// TIA Portal V15.1 export
// export: Created 2024-05-17T05:38:52.2230913Z, ExportSetting WithDefaults, DisplayName Totally Integrated Automation Portal, DisplayVersion V15.1 Update 5, DisplayName TIA Portal Openness, DisplayVersion V15.1 Update 5, DisplayName SINAMICS Startdrive Advanced, DisplayVersion V15.1, DisplayName G130, G150, S120, S150, SINAMICS MV, S210, DisplayVersion V15.1, DisplayName G110M, G120, G120C, G120D, G120P, DisplayVersion V15.1, DisplayName STEP 7 Professional, DisplayVersion V15.1 Update 5, DisplayName STEP 7 Safety, DisplayVersion V15.1, DisplayName WinCC Professional, DisplayVersion V15.1 Update 5, DisplayName SIMATIC Visualization Architect, DisplayVersion V15.1
FUNCTION_BLOCK "LGBShuttle5Pos2S-MoviFitFCPN"   // FB6696, FBD
TITLE = LGBFlinta5Pos3S-MoviFitFCPN / LGBShuttle5Pos2S-MoviFitFCPN
{ S7_Optimized_Access := 'TRUE' }
AUTHOR : VCC
VERSION : 0.0.0.0
// stored: AutoNumber false, IsIECCheckEnabled false, IsRetainMemResEnabled false, MemoryReserve 100, SetENOAutomatically False, UDAEnableTagReadback false
   VAR_INPUT
      I_Position1Begin { ExternalAccessible := 'False'; ExternalVisible := 'False'; ExternalWritable := 'False'} : Bool;   // Start Move To Position / Start Move To Position 1
      I_Position2Begin { ExternalAccessible := 'False'; ExternalVisible := 'False'; ExternalWritable := 'False'} : Bool;   // Start Move To Position / Start Move To Position 2
      I_Position3Begin { ExternalAccessible := 'False'; ExternalVisible := 'False'; ExternalWritable := 'False'} : Bool;   // Start Move To Position / Start Move To Position 3
      I_Position4Begin { ExternalAccessible := 'False'; ExternalVisible := 'False'; ExternalWritable := 'False'} : Bool;   // Start Move To Position / Start Move To Position 4
      I_Position5Begin { ExternalAccessible := 'False'; ExternalVisible := 'False'; ExternalWritable := 'False'} : Bool;   // Start Move To Position / Start Move To Position 5
      I_PositionMaintBegin { ExternalAccessible := 'False'; ExternalVisible := 'False'; ExternalWritable := 'False'} : Bool;   // Start Move To Position Maintenance
      I_SetIntlkOK { ExternalAccessible := 'False'; ExternalVisible := 'False'; ExternalWritable := 'False'} : Bool;   // Set Interlock
      I_ResIntlkOK { ExternalAccessible := 'False'; ExternalVisible := 'False'; ExternalWritable := 'False'} : Bool;   // Reset Interlock
      I_LocalPBSet { ExternalAccessible := 'False'; ExternalVisible := 'False'; ExternalWritable := 'False'} : Bool;   // Push button for manual movememt Set (on local panel)
      I_LocalPBRes { ExternalAccessible := 'False'; ExternalVisible := 'False'; ExternalWritable := 'False'} : Bool;   // Push button for manual movememt Reset (on local panel)
      I_MotorProtection { ExternalAccessible := 'False'; ExternalVisible := 'False'; ExternalWritable := 'False'} : Bool;   // Motor protection
      I_HartingPlug400V { ExternalAccessible := 'False'; ExternalVisible := 'False'; ExternalWritable := 'False'} : Bool;   // Harting plug 400V
      I_HartingPlug24V { ExternalAccessible := 'False'; ExternalVisible := 'False'; ExternalWritable := 'False'} : Bool;   // Harting plug 24V
      I_OvertravelSet { ExternalAccessible := 'False'; ExternalVisible := 'False'; ExternalWritable := 'False'} : Bool;   // Overtravel Set
      I_OvertravelRes { ExternalAccessible := 'False'; ExternalVisible := 'False'; ExternalWritable := 'False'} : Bool;   // Overtravel Reset
      I_ReferenceDet { ExternalAccessible := 'False'; ExternalVisible := 'False'; ExternalWritable := 'False'} : Bool;   // Reference detection
      I_ReleaseBrake { ExternalAccessible := 'False'; ExternalVisible := 'False'; ExternalWritable := 'False'} : Bool;   // Release brake
      I_Distance { ExternalAccessible := 'False'; ExternalVisible := 'False'; ExternalWritable := 'False'} : DInt;   // Current distance
      I_SafetyOk { ExternalAccessible := 'False'; ExternalVisible := 'False'; ExternalWritable := 'False'} : Bool;   // Safety Ok
      I_MotionStopOk { ExternalAccessible := 'False'; ExternalVisible := 'False'; ExternalWritable := 'False'} : Bool;   // The motion stop is Ok
      I_LowSpeed { ExternalAccessible := 'False'; ExternalVisible := 'False'; ExternalWritable := 'False'} : Real;   // Low speed Value (set-up %)
      I_HighSpeed { ExternalAccessible := 'False'; ExternalVisible := 'False'; ExternalWritable := 'False'} : Real;   // High speed Value (set-up %)
      I_SafetyStatusWord { ExternalAccessible := 'False'; ExternalVisible := 'False'; ExternalWritable := 'False'} : Word;   // Safety Status
      I_SafetyControlWord { ExternalAccessible := 'False'; ExternalVisible := 'False'; ExternalWritable := 'False'} : Word;   // Safety Control Word
   END_VAR
   VAR_OUTPUT
      O_ReleaseBrake { ExternalAccessible := 'False'; ExternalVisible := 'False'; ExternalWritable := 'False'} : Bool;   // Release the brake of the Motor
      O_Active { ExternalAccessible := 'False'; ExternalVisible := 'False'; ExternalWritable := 'False'} : Bool;   // Machine is active
      O_FuncRunning { ExternalAccessible := 'False'; ExternalVisible := 'False'; ExternalWritable := 'False'} : Bool;   // Signal that the function is busy
      O_InPosition1 { ExternalAccessible := 'False'; ExternalVisible := 'False'; ExternalWritable := 'False'} : Bool;   // In Position 1
      O_InPosition2 { ExternalAccessible := 'False'; ExternalVisible := 'False'; ExternalWritable := 'False'} : Bool;   // In Position 2
      O_InPosition3 { ExternalAccessible := 'False'; ExternalVisible := 'False'; ExternalWritable := 'False'} : Bool;   // In Position 3
      O_InPosition4 { ExternalAccessible := 'False'; ExternalVisible := 'False'; ExternalWritable := 'False'} : Bool;   // In Position 4
      O_InPosition5 { ExternalAccessible := 'False'; ExternalVisible := 'False'; ExternalWritable := 'False'} : Bool;   // In Position 5
      O_InPositionMaint { ExternalAccessible := 'False'; ExternalVisible := 'False'; ExternalWritable := 'False'} : Bool;   // In Position Maintenance
      O_Position1Finished { ExternalAccessible := 'False'; ExternalVisible := 'False'; ExternalWritable := 'False'} : Bool;   // Position 1 finished
      O_Position2Finished { ExternalAccessible := 'False'; ExternalVisible := 'False'; ExternalWritable := 'False'} : Bool;   // Position 2 finished
      O_Position3Finished { ExternalAccessible := 'False'; ExternalVisible := 'False'; ExternalWritable := 'False'} : Bool;   // Position 3 finished
      O_Position4Finished { ExternalAccessible := 'False'; ExternalVisible := 'False'; ExternalWritable := 'False'} : Bool;   // Position 4 finished
      O_Position5Finished { ExternalAccessible := 'False'; ExternalVisible := 'False'; ExternalWritable := 'False'} : Bool;   // Position 5 finished
      O_PositionMaintFinished { ExternalAccessible := 'False'; ExternalVisible := 'False'; ExternalWritable := 'False'} : Bool;   // Position Maintenance finished
      O_LEDPosition1 { ExternalAccessible := 'False'; ExternalVisible := 'False'; ExternalWritable := 'False'} : Bool;   // Ledindication / Led indication for Position1
      O_LEDPosition2 { ExternalAccessible := 'False'; ExternalVisible := 'False'; ExternalWritable := 'False'} : Bool;   // Ledindication / Led indication for Position2
      O_LEDPosition3 { ExternalAccessible := 'False'; ExternalVisible := 'False'; ExternalWritable := 'False'} : Bool;   // Ledindication / Led indication for Position3
      O_LEDPosition4 { ExternalAccessible := 'False'; ExternalVisible := 'False'; ExternalWritable := 'False'} : Bool;   // Ledindication / Led indication for Position4
      O_LEDPosition5 { ExternalAccessible := 'False'; ExternalVisible := 'False'; ExternalWritable := 'False'} : Bool;   // Ledindication / Led indication for Position5
      O_ReadyForOperation { ExternalAccessible := 'False'; ExternalVisible := 'False'; ExternalWritable := 'False'} : Bool;   // Ready for operation
      O_AlarmABCondition { ExternalAccessible := 'False'; ExternalVisible := 'False'; ExternalWritable := 'False'} : Bool;   // Alarm AB condition
      O_AlarmA { ExternalAccessible := 'False'; ExternalVisible := 'False'; ExternalWritable := 'False'} : Bool;   // Summation Alarm A
      O_AlarmB { ExternalAccessible := 'False'; ExternalVisible := 'False'; ExternalWritable := 'False'} : Bool;   // Summation Alarm B
      O_AlarmC { ExternalAccessible := 'False'; ExternalVisible := 'False'; ExternalWritable := 'False'} : Bool;   // Summation Alarm C
      O_AlarmD { ExternalAccessible := 'False'; ExternalVisible := 'False'; ExternalWritable := 'False'} : Bool;   // Summation Alarm D
      H_AlarmDWord { ExternalAccessible := 'False'; ExternalVisible := 'False'; ExternalWritable := 'False'} : DWord;   // HMI Animation of the alarms
      H_ActPosShuttle { ExternalAccessible := 'False'; ExternalVisible := 'False'; ExternalWritable := 'False'} : Int;   // HMI Animation Position of the Shuttle
   END_VAR
   VAR_IN_OUT
      IO_Modes : "Modes";   // Modes
      H_HMI : "H_HMI";   // Animation
      "H_GBShuttle5Pos2S-MoviFitFCPN" : "H_GBShuttle5Pos2S-MoviFitFCPN";   // Animation
      C_Config : "Shuttle5Pos2S-MoviFitFCPNConfig";   // Config
   END_VAR
   VAR
      AA_MotorProtection { ExternalAccessible := 'False'; ExternalVisible := 'False'; ExternalWritable := 'False'} : Bool;   // Motorprotection Not Ok
      AA_SafetySwitch { ExternalAccessible := 'False'; ExternalVisible := 'False'; ExternalWritable := 'False'} : Bool;   // Safety Switch Not Ok
      AB_STO { ExternalAccessible := 'False'; ExternalVisible := 'False'; ExternalWritable := 'False'} : Bool;   // Safety Switch Not Ok / Safety output to drive is active but no response from drive that the safety is ok
      AB_DriveAlarm { ExternalAccessible := 'False'; ExternalVisible := 'False'; ExternalWritable := 'False'} : Bool;   // Alarm Frequency Control
      AB_OverTravelSet { ExternalAccessible := 'False'; ExternalVisible := 'False'; ExternalWritable := 'False'} : Bool;   // Overtravel Set
      AB_OverTravelRes { ExternalAccessible := 'False'; ExternalVisible := 'False'; ExternalWritable := 'False'} : Bool;   // Overtravel Reset
      AC_KeepPos1 { ExternalAccessible := 'False'; ExternalVisible := 'False'; ExternalWritable := 'False'} : Bool;   // Lost Position 1
      AC_KeepPos2 { ExternalAccessible := 'False'; ExternalVisible := 'False'; ExternalWritable := 'False'} : Bool;   // Lost Position 2
      AC_KeepPos3 { ExternalAccessible := 'False'; ExternalVisible := 'False'; ExternalWritable := 'False'} : Bool;   // Lost Position 3
      AC_KeepPos4 { ExternalAccessible := 'False'; ExternalVisible := 'False'; ExternalWritable := 'False'} : Bool;   // Lost Position 4
      AC_KeepPos5 { ExternalAccessible := 'False'; ExternalVisible := 'False'; ExternalWritable := 'False'} : Bool;   // Lost Position 5
      AC_OvtSetAlm { ExternalAccessible := 'False'; ExternalVisible := 'False'; ExternalWritable := 'False'} : Bool;   // Timeout Set / TimeOut Set Direction
      AC_OvtResAlm { ExternalAccessible := 'False'; ExternalVisible := 'False'; ExternalWritable := 'False'} : Bool;   // Timeout Reset / TimeOut Reset Direction
      AD_IntlkSetAlm { ExternalAccessible := 'False'; ExternalVisible := 'False'; ExternalWritable := 'False'} : Bool;   // Interlock Set
      AD_IntlkResAlm { ExternalAccessible := 'False'; ExternalVisible := 'False'; ExternalWritable := 'False'} : Bool;   // Interlock Reset
      AD_OvtSetWarn { ExternalAccessible := 'False'; ExternalVisible := 'False'; ExternalWritable := 'False'} : Bool;   // TimeOut Set Direction
      AD_OvtResWarn { ExternalAccessible := 'False'; ExternalVisible := 'False'; ExternalWritable := 'False'} : Bool;   // TimeOut Reset Direction
      AD_DriveWarning { ExternalAccessible := 'False'; ExternalVisible := 'False'; ExternalWritable := 'False'} : Bool;   // Warning Frequency Control
      AA_NoBusControl { ExternalAccessible := 'False'; ExternalVisible := 'False'; ExternalWritable := 'False'} : Bool;   // Bus Control Inactive Frequency Control
      AA_HartingPlug400V { ExternalAccessible := 'False'; ExternalVisible := 'False'; ExternalWritable := 'False'} : Bool;   // Harting plug MoviFits 400VAC Not Ok
      AA_HartingPlug24V { ExternalAccessible := 'False'; ExternalVisible := 'False'; ExternalWritable := 'False'} : Bool;   // Harting plug MoviFits 24VDC Not Ok
      AB_ReferencingMode { ExternalAccessible := 'False'; ExternalVisible := 'False'; ExternalWritable := 'False'} : Bool;   // Shuttle in Referencing Mode / Flinta in Referencing Mode
      AB_NoReferencing { ExternalAccessible := 'False'; ExternalVisible := 'False'; ExternalWritable := 'False'} : Bool;   // The referencing of the Shuttle is not done. Start the Referencing procedure!
      AD_MotionStop { ExternalAccessible := 'False'; ExternalVisible := 'False'; ExternalWritable := 'False'} : Bool;   // Motion Stop
      AC_ConfigCalibrationAlm { ExternalAccessible := 'False'; ExternalVisible := 'False'; ExternalWritable := 'False'} : Bool;   // The Config values for Warming/Alarm time must be ALL zero or ALL different from zero
      AD_CalibrationWarn { ExternalAccessible := 'False'; ExternalVisible := 'False'; ExternalWritable := 'False'} : Bool;   // No High speed selected so Calibration is not possible
      AC_ConfigRampAlm { ExternalAccessible := 'False'; ExternalVisible := 'False'; ExternalWritable := 'False'} : Bool;   // The config value for the ramp is not correct, must be zero or the config values for the calculation of the ramp must be ALL zero
      AC_ConfigRampCalcAlm { ExternalAccessible := 'False'; ExternalVisible := 'False'; ExternalWritable := 'False'} : Bool;   // The config values for the calculation of the ramp must be ALL different from zero
      AD_ReferencingActive { ExternalAccessible := 'False'; ExternalVisible := 'False'; ExternalWritable := 'False'} : Bool;   // Referencing is active
      SafetyOk { ExternalAccessible := 'False'; ExternalVisible := 'False'; ExternalWritable := 'False'} : Bool;   // Safety Ok
      AlarmA { ExternalAccessible := 'False'; ExternalVisible := 'False'; ExternalWritable := 'False'} : Bool;   // Alarm A
      AlarmB { ExternalAccessible := 'False'; ExternalVisible := 'False'; ExternalWritable := 'False'} : Bool;   // Alarm B
      AlarmC { ExternalAccessible := 'False'; ExternalVisible := 'False'; ExternalWritable := 'False'} : Bool;   // Alarm C
      AlarmD { ExternalAccessible := 'False'; ExternalVisible := 'False'; ExternalWritable := 'False'} : Bool;   // Alarm D
      AlarmABCondition { ExternalAccessible := 'False'; ExternalVisible := 'False'; ExternalWritable := 'False'} : Bool;   // Alarm AB Condition
      RunTimeMaxWarn { ExternalAccessible := 'False'; ExternalVisible := 'False'; ExternalWritable := 'False'} : DInt;   // Maximum run time warning
      RunTimeMaxAlm { ExternalAccessible := 'False'; ExternalVisible := 'False'; ExternalWritable := 'False'} : DInt;   // Maximum run time alarm
      RunTimeMaxSetWarn { ExternalAccessible := 'False'; ExternalVisible := 'False'; ExternalWritable := 'False'} : DInt;   // Maximum run time warning
      RunTimeMaxSetAlm { ExternalAccessible := 'False'; ExternalVisible := 'False'; ExternalWritable := 'False'} : DInt;   // Maximum run time alarm
      RunTimeMaxResWarn { ExternalAccessible := 'False'; ExternalVisible := 'False'; ExternalWritable := 'False'} : DInt;   // Maximum run time warning
      RunTimeMaxResAlm { ExternalAccessible := 'False'; ExternalVisible := 'False'; ExternalWritable := 'False'} : DInt;   // Maximum run time alarm
      MovFuncAlmCond { ExternalAccessible := 'False'; ExternalVisible := 'False'; ExternalWritable := 'False'} : Bool;   // Move function Alarm Condition
      StopPosAlmCond { ExternalAccessible := 'False'; ExternalVisible := 'False'; ExternalWritable := 'False'} : Bool;   // Stop posistion Alarm Condition
      MotorLoopActive { ExternalAccessible := 'False'; ExternalVisible := 'False'; ExternalWritable := 'False'} : Bool;   // Motor Loop Active
      OverTravelSetAlmCond { ExternalAccessible := 'False'; ExternalVisible := 'False'; ExternalWritable := 'False'} : Bool;   // Overtravel set alarm condition
      OverTravelResAlmCond { ExternalAccessible := 'False'; ExternalVisible := 'False'; ExternalWritable := 'False'} : Bool;   // Overtravel reset alarm condition
      HartingPlug400VAlmCond { ExternalAccessible := 'False'; ExternalVisible := 'False'; ExternalWritable := 'False'} : Bool;   // Harting plug 400V alarm condition
      HartingPlug24VAlmCond { ExternalAccessible := 'False'; ExternalVisible := 'False'; ExternalWritable := 'False'} : Bool;   // Harting plug 24V alarm condition
      FuncRunning { ExternalAccessible := 'False'; ExternalVisible := 'False'; ExternalWritable := 'False'} : Bool;   // Function running
      CmdSet { ExternalAccessible := 'False'; ExternalVisible := 'False'; ExternalWritable := 'False'} : Bool;   // Command set
      CmdRes { ExternalAccessible := 'False'; ExternalVisible := 'False'; ExternalWritable := 'False'} : Bool;   // DCommand Reset
      MotorLoopAlarmCond { ExternalAccessible := 'False'; ExternalVisible := 'False'; ExternalWritable := 'False'} : Bool;   // Motor loop alarm condition
      LowerLimit { ExternalAccessible := 'False'; ExternalVisible := 'False'; ExternalWritable := 'False'} : DInt;   // Lowest position
      UpperLimit { ExternalAccessible := 'False'; ExternalVisible := 'False'; ExternalWritable := 'False'} : DInt;   // Highest position
      DiffPos { ExternalAccessible := 'False'; ExternalVisible := 'False'; ExternalWritable := 'False'} : DInt;   // Diff position
      ReferencingMode { ExternalAccessible := 'False'; ExternalVisible := 'False'; ExternalWritable := 'False'} : Bool;   // Referencing Mode
      ReferencingOvertravel { ExternalAccessible := 'False'; ExternalVisible := 'False'; ExternalWritable := 'False'} : Bool;   // During referencing mode is overtravel reached
      ReferencingFinished { ExternalAccessible := 'False'; ExternalVisible := 'False'; ExternalWritable := 'False'} : Bool;   // Referencing mode is finished
      CalculatedPos1 { ExternalAccessible := 'False'; ExternalVisible := 'False'; ExternalWritable := 'False'} : DInt;   // Calculated position 1
      CalculatedPos2 { ExternalAccessible := 'False'; ExternalVisible := 'False'; ExternalWritable := 'False'} : DInt;   // Calculated position 2
      CalculatedPos3 { ExternalAccessible := 'False'; ExternalVisible := 'False'; ExternalWritable := 'False'} : DInt;   // Calculated position 3
      CalculatedPos4 { ExternalAccessible := 'False'; ExternalVisible := 'False'; ExternalWritable := 'False'} : DInt;   // Calculated position 4
      CalculatedPos5 { ExternalAccessible := 'False'; ExternalVisible := 'False'; ExternalWritable := 'False'} : DInt;   // Calculated position 5
      CalculatedPosMaint { ExternalAccessible := 'False'; ExternalVisible := 'False'; ExternalWritable := 'False'} : DInt;   // Calculated Maintenance Position
      DirectionSetPos1 { ExternalAccessible := 'False'; ExternalVisible := 'False'; ExternalWritable := 'False'} : Bool;   // Direction SET position 1
      DirectionSetPos2 { ExternalAccessible := 'False'; ExternalVisible := 'False'; ExternalWritable := 'False'} : Bool;   // Direction SET position 2
      DirectionSetPos3 { ExternalAccessible := 'False'; ExternalVisible := 'False'; ExternalWritable := 'False'} : Bool;   // Direction SET position 3
      DirectionSetPos4 { ExternalAccessible := 'False'; ExternalVisible := 'False'; ExternalWritable := 'False'} : Bool;   // Direction SET position 4
      DirectionSetPos5 { ExternalAccessible := 'False'; ExternalVisible := 'False'; ExternalWritable := 'False'} : Bool;   // Direction SET position 5
      DirectionSetPosMaint { ExternalAccessible := 'False'; ExternalVisible := 'False'; ExternalWritable := 'False'} : Bool;   // Direction SET position Maintenance
      DirectionResPos1 { ExternalAccessible := 'False'; ExternalVisible := 'False'; ExternalWritable := 'False'} : Bool;   // Direction RESET position 1
      DirectionResPos2 { ExternalAccessible := 'False'; ExternalVisible := 'False'; ExternalWritable := 'False'} : Bool;   // Direction RESET position 2
      DirectionResPos3 { ExternalAccessible := 'False'; ExternalVisible := 'False'; ExternalWritable := 'False'} : Bool;   // Direction RESET position 3
      DirectionResPos4 { ExternalAccessible := 'False'; ExternalVisible := 'False'; ExternalWritable := 'False'} : Bool;   // Direction RESET position 4
      DirectionResPos5 { ExternalAccessible := 'False'; ExternalVisible := 'False'; ExternalWritable := 'False'} : Bool;   // Direction RESET position 5
      DirectionResPosMaint { ExternalAccessible := 'False'; ExternalVisible := 'False'; ExternalWritable := 'False'} : Bool;   // Direction RESET position Maintenance
      ManReqSetPos1 { ExternalAccessible := 'False'; ExternalVisible := 'False'; ExternalWritable := 'False'} : Bool;   // Manual request SET position 1
      ManReqSetPos2 { ExternalAccessible := 'False'; ExternalVisible := 'False'; ExternalWritable := 'False'} : Bool;   // Manual request SET position 2
      ManReqSetPos3 { ExternalAccessible := 'False'; ExternalVisible := 'False'; ExternalWritable := 'False'} : Bool;   // Manual request SET position 3
      ManReqSetPos4 { ExternalAccessible := 'False'; ExternalVisible := 'False'; ExternalWritable := 'False'} : Bool;   // Manual request SET position 4
      ManReqSetPos5 { ExternalAccessible := 'False'; ExternalVisible := 'False'; ExternalWritable := 'False'} : Bool;   // Manual request SET position 5
      ManReqSetPosMaint { ExternalAccessible := 'False'; ExternalVisible := 'False'; ExternalWritable := 'False'} : Bool;   // Manual request SET position Maintenance
      ManReqResPos1 { ExternalAccessible := 'False'; ExternalVisible := 'False'; ExternalWritable := 'False'} : Bool;   // Manual request RESET position 1
      ManReqResPos2 { ExternalAccessible := 'False'; ExternalVisible := 'False'; ExternalWritable := 'False'} : Bool;   // Manual request RESET position 2
      ManReqResPos3 { ExternalAccessible := 'False'; ExternalVisible := 'False'; ExternalWritable := 'False'} : Bool;   // Manual request RESET position 3
      ManReqResPos4 { ExternalAccessible := 'False'; ExternalVisible := 'False'; ExternalWritable := 'False'} : Bool;   // Manual request RESET position 4
      ManReqResPos5 { ExternalAccessible := 'False'; ExternalVisible := 'False'; ExternalWritable := 'False'} : Bool;   // Manual request RESET position 5
      ManReqResPosMaint { ExternalAccessible := 'False'; ExternalVisible := 'False'; ExternalWritable := 'False'} : Bool;   // Manual request RESET position Maintenance
      AutoReqSetPos1 { ExternalAccessible := 'False'; ExternalVisible := 'False'; ExternalWritable := 'False'} : Bool;   // Auto request SET position 1
      AutoReqSetPos2 { ExternalAccessible := 'False'; ExternalVisible := 'False'; ExternalWritable := 'False'} : Bool;   // Auto request SET position 2
      AutoReqSetPos3 { ExternalAccessible := 'False'; ExternalVisible := 'False'; ExternalWritable := 'False'} : Bool;   // Auto request SET position 3
      AutoReqSetPos4 { ExternalAccessible := 'False'; ExternalVisible := 'False'; ExternalWritable := 'False'} : Bool;   // Auto request SET position 4
      AutoReqSetPos5 { ExternalAccessible := 'False'; ExternalVisible := 'False'; ExternalWritable := 'False'} : Bool;   // Auto request SET position 5
      AutoReqSetPosMaint { ExternalAccessible := 'False'; ExternalVisible := 'False'; ExternalWritable := 'False'} : Bool;   // Auto request SET position Maintenance
      AutoReqResPos1 { ExternalAccessible := 'False'; ExternalVisible := 'False'; ExternalWritable := 'False'} : Bool;   // Auto request RESET position 1
      AutoReqResPos2 { ExternalAccessible := 'False'; ExternalVisible := 'False'; ExternalWritable := 'False'} : Bool;   // Auto request RESET position 2
      AutoReqResPos3 { ExternalAccessible := 'False'; ExternalVisible := 'False'; ExternalWritable := 'False'} : Bool;   // Auto request RESET position 3
      AutoReqResPos4 { ExternalAccessible := 'False'; ExternalVisible := 'False'; ExternalWritable := 'False'} : Bool;   // Auto request RESET position 4
      AutoReqResPos5 { ExternalAccessible := 'False'; ExternalVisible := 'False'; ExternalWritable := 'False'} : Bool;   // Auto request RESET position 5
      AutoReqResPosMaint { ExternalAccessible := 'False'; ExternalVisible := 'False'; ExternalWritable := 'False'} : Bool;   // Auto request RESET position Maintenance
      CmdSetPos1 { ExternalAccessible := 'False'; ExternalVisible := 'False'; ExternalWritable := 'False'} : Bool;   // Command to Position 1 in SET
      CmdSetPos2 { ExternalAccessible := 'False'; ExternalVisible := 'False'; ExternalWritable := 'False'} : Bool;   // Command to Position 2 in SET
      CmdSetPos3 { ExternalAccessible := 'False'; ExternalVisible := 'False'; ExternalWritable := 'False'} : Bool;   // Command to Position 3 in SET
      CmdSetPos4 { ExternalAccessible := 'False'; ExternalVisible := 'False'; ExternalWritable := 'False'} : Bool;   // Command to Position 4 in SET
      CmdSetPos5 { ExternalAccessible := 'False'; ExternalVisible := 'False'; ExternalWritable := 'False'} : Bool;   // Command to Position 5 in SET
      CmdSetPosMaint { ExternalAccessible := 'False'; ExternalVisible := 'False'; ExternalWritable := 'False'} : Bool;   // Command to Position Maintenance in SET
      CmdResPos1 { ExternalAccessible := 'False'; ExternalVisible := 'False'; ExternalWritable := 'False'} : Bool;   // Command to Position 1 in RESET
      CmdResPos2 { ExternalAccessible := 'False'; ExternalVisible := 'False'; ExternalWritable := 'False'} : Bool;   // Command to Position 2 in RESET
      CmdResPos3 { ExternalAccessible := 'False'; ExternalVisible := 'False'; ExternalWritable := 'False'} : Bool;   // Command to Position 3 in RESET
      CmdResPos4 { ExternalAccessible := 'False'; ExternalVisible := 'False'; ExternalWritable := 'False'} : Bool;   // Command to Position 4 in RESET
      CmdResPos5 { ExternalAccessible := 'False'; ExternalVisible := 'False'; ExternalWritable := 'False'} : Bool;   // Command to Position 5 in RESET
      CmdResPosMaint { ExternalAccessible := 'False'; ExternalVisible := 'False'; ExternalWritable := 'False'} : Bool;   // Command to Position Maintenance in RESET
      CmdPos1 { ExternalAccessible := 'False'; ExternalVisible := 'False'; ExternalWritable := 'False'} : Bool;   // Command to Position 1
      CmdPos2 { ExternalAccessible := 'False'; ExternalVisible := 'False'; ExternalWritable := 'False'} : Bool;   // Command to Position 2
      CmdPos3 { ExternalAccessible := 'False'; ExternalVisible := 'False'; ExternalWritable := 'False'} : Bool;   // Command to Position 3
      CmdPos4 { ExternalAccessible := 'False'; ExternalVisible := 'False'; ExternalWritable := 'False'} : Bool;   // Command to Position 4
      CmdPos5 { ExternalAccessible := 'False'; ExternalVisible := 'False'; ExternalWritable := 'False'} : Bool;   // Command to Position 5
      CmdPosMaint { ExternalAccessible := 'False'; ExternalVisible := 'False'; ExternalWritable := 'False'} : Bool;   // Command to Position Maintenance
      Pos1IsHomePos { ExternalAccessible := 'False'; ExternalVisible := 'False'; ExternalWritable := 'False'} : Bool;   // In position 1 / Position 1 is home position
      Pos2IsHomePos { ExternalAccessible := 'False'; ExternalVisible := 'False'; ExternalWritable := 'False'} : Bool;   // In position 2 / Position 2 is home position
      Pos3IsHomePos { ExternalAccessible := 'False'; ExternalVisible := 'False'; ExternalWritable := 'False'} : Bool;   // In position 3 / Position 3 is home position
      Pos4IsHomePos { ExternalAccessible := 'False'; ExternalVisible := 'False'; ExternalWritable := 'False'} : Bool;   // In position 4 / Position 4 is home position
      Pos5IsHomePos { ExternalAccessible := 'False'; ExternalVisible := 'False'; ExternalWritable := 'False'} : Bool;   // In position 5 / Position 5 is home position
      InPos1 { ExternalAccessible := 'False'; ExternalVisible := 'False'; ExternalWritable := 'False'} : Bool;   // In position 1
      InPos2 { ExternalAccessible := 'False'; ExternalVisible := 'False'; ExternalWritable := 'False'} : Bool;   // In position 2
      InPos3 { ExternalAccessible := 'False'; ExternalVisible := 'False'; ExternalWritable := 'False'} : Bool;   // In position 3
      InPos4 { ExternalAccessible := 'False'; ExternalVisible := 'False'; ExternalWritable := 'False'} : Bool;   // In position 4
      InPos5 { ExternalAccessible := 'False'; ExternalVisible := 'False'; ExternalWritable := 'False'} : Bool;   // In position 5
      InPosMaint { ExternalAccessible := 'False'; ExternalVisible := 'False'; ExternalWritable := 'False'} : Bool;   // In position Maintenance
      SetIntlkOK { ExternalAccessible := 'False'; ExternalVisible := 'False'; ExternalWritable := 'False'} : Bool;   // Interlock Pos1
      ResIntlkOK { ExternalAccessible := 'False'; ExternalVisible := 'False'; ExternalWritable := 'False'} : Bool;   // Interlock Pos2
      ReadyForOperation { ExternalAccessible := 'False'; ExternalVisible := 'False'; ExternalWritable := 'False'} : Bool;   // Ready for operation
      LastCmd1 { ExternalAccessible := 'False'; ExternalVisible := 'False'; ExternalWritable := 'False'} : Bool;   // Last Command to Drive Is Pos 1
      LastCmd2 { ExternalAccessible := 'False'; ExternalVisible := 'False'; ExternalWritable := 'False'} : Bool;   // Last Command to Drive Is Pos 2
      LastCmd3 { ExternalAccessible := 'False'; ExternalVisible := 'False'; ExternalWritable := 'False'} : Bool;   // Last Command to Drive Is Pos 3
      LastCmd4 { ExternalAccessible := 'False'; ExternalVisible := 'False'; ExternalWritable := 'False'} : Bool;   // Last Command to Drive Is Pos 4
      LastCmd5 { ExternalAccessible := 'False'; ExternalVisible := 'False'; ExternalWritable := 'False'} : Bool;   // Last Command to Drive Is Pos 5
      AlmCondKeepPos1 { ExternalAccessible := 'False'; ExternalVisible := 'False'; ExternalWritable := 'False'} : Bool;   // Alarm Condition Keep Position 1
      AlmCondKeepPos2 { ExternalAccessible := 'False'; ExternalVisible := 'False'; ExternalWritable := 'False'} : Bool;   // Alarm Condition Keep Position 2
      AlmCondKeepPos3 { ExternalAccessible := 'False'; ExternalVisible := 'False'; ExternalWritable := 'False'} : Bool;   // Alarm Condition Keep Position 3
      AlmCondKeepPos4 { ExternalAccessible := 'False'; ExternalVisible := 'False'; ExternalWritable := 'False'} : Bool;   // Alarm Condition Keep Position 4
      AlmCondKeepPos5 { ExternalAccessible := 'False'; ExternalVisible := 'False'; ExternalWritable := 'False'} : Bool;   // Alarm Condition Keep Position 5
      DetLowSpeedPos1 { ExternalAccessible := 'False'; ExternalVisible := 'False'; ExternalWritable := 'False'} : Bool;   // Stop high speed
      DetStopPos1 { ExternalAccessible := 'False'; ExternalVisible := 'False'; ExternalWritable := 'False'} : Bool;   // Stop on position
      DetLowSpeedPos2 { ExternalAccessible := 'False'; ExternalVisible := 'False'; ExternalWritable := 'False'} : Bool;   // Stop high speed
      DetStopPos2 { ExternalAccessible := 'False'; ExternalVisible := 'False'; ExternalWritable := 'False'} : Bool;   // Stop on position
      DetLowSpeedPos3 { ExternalAccessible := 'False'; ExternalVisible := 'False'; ExternalWritable := 'False'} : Bool;   // Stop high speed
      DetStopPos3 { ExternalAccessible := 'False'; ExternalVisible := 'False'; ExternalWritable := 'False'} : Bool;   // Stop on position
      DetLowSpeedPos4 { ExternalAccessible := 'False'; ExternalVisible := 'False'; ExternalWritable := 'False'} : Bool;   // Stop high speed
      DetStopPos4 { ExternalAccessible := 'False'; ExternalVisible := 'False'; ExternalWritable := 'False'} : Bool;   // Stop on position
      DetLowSpeedPos5 { ExternalAccessible := 'False'; ExternalVisible := 'False'; ExternalWritable := 'False'} : Bool;   // Stop high speed
      DetStopPos5 { ExternalAccessible := 'False'; ExternalVisible := 'False'; ExternalWritable := 'False'} : Bool;   // Stop on position
      DetLowSpeedPosMaint { ExternalAccessible := 'False'; ExternalVisible := 'False'; ExternalWritable := 'False'} : Bool;   // Stop high speed
      DetStopPosMaint { ExternalAccessible := 'False'; ExternalVisible := 'False'; ExternalWritable := 'False'} : Bool;   // Stop on position
      LockLocalPB { ExternalAccessible := 'False'; ExternalVisible := 'False'; ExternalWritable := 'False'} : Bool;   // Lock push button
      PODataNotEnabled { ExternalAccessible := 'False'; ExternalVisible := 'False'; ExternalWritable := 'False'} : Bool;   // Bus control inactive
      ReleaseBrake { ExternalAccessible := 'False'; ExternalVisible := 'False'; ExternalWritable := 'False'} : Bool;   // Release brake
      MotorCmdLSpdSet { ExternalAccessible := 'False'; ExternalVisible := 'False'; ExternalWritable := 'False'} : Bool;   // Command to Motorloop low Speed Set
      MotorCmdLSpdRes { ExternalAccessible := 'False'; ExternalVisible := 'False'; ExternalWritable := 'False'} : Bool;   // Command to Motorloop low speed Reset
      MotorCmdHSpdSet { ExternalAccessible := 'False'; ExternalVisible := 'False'; ExternalWritable := 'False'} : Bool;   // Command to Motorloop High Speed Set
      MotorCmdHSpdRes { ExternalAccessible := 'False'; ExternalVisible := 'False'; ExternalWritable := 'False'} : Bool;   // Command to Motorloop High Speed Reset
      PosSet { ExternalAccessible := 'False'; ExternalVisible := 'False'; ExternalWritable := 'False'} : Bool;   // Position Set detection or summary
      LowSpeedSetDet { ExternalAccessible := 'False'; ExternalVisible := 'False'; ExternalWritable := 'False'} : Bool;   // Slow Set detection or summary
      PosRes { ExternalAccessible := 'False'; ExternalVisible := 'False'; ExternalWritable := 'False'} : Bool;   // Position Reset detection or summary
      LowSpeedResDet { ExternalAccessible := 'False'; ExternalVisible := 'False'; ExternalWritable := 'False'} : Bool;   // Slow Reset detection or summary
      SetBegin { ExternalAccessible := 'False'; ExternalVisible := 'False'; ExternalWritable := 'False'} : Bool;   // Function Set begin selection
      ResBegin { ExternalAccessible := 'False'; ExternalVisible := 'False'; ExternalWritable := 'False'} : Bool;   // Function Reset begin selection
      InitDirection { ExternalAccessible := 'False'; ExternalVisible := 'False'; ExternalWritable := 'False'} : Bool;   // Initialisation of the direction
      LowSpeed { ExternalAccessible := 'False'; ExternalVisible := 'False'; ExternalWritable := 'False'} : Real;   // Low speed Value (set-up %)
      H_FncSelInHMI { ExternalAccessible := 'False'; ExternalVisible := 'False'; ExternalWritable := 'False'} : Bool;   // Function select
      H_ReferencingMode { ExternalAccessible := 'False'; ExternalVisible := 'False'; ExternalWritable := 'False'} : Bool;   // HMI Command - Activate referencing
      H_ReferencingAccept { ExternalAccessible := 'False'; ExternalVisible := 'False'; ExternalWritable := 'False'} : Bool;   // HMI Command - Reference button to accept new values
      H_CmdPos1 { ExternalAccessible := 'False'; ExternalVisible := 'False'; ExternalWritable := 'False'} : Bool;   // HMI Command - To Pos1
      H_CmdPos2 { ExternalAccessible := 'False'; ExternalVisible := 'False'; ExternalWritable := 'False'} : Bool;   // HMI Command - To Pos2
      H_CmdPos3 { ExternalAccessible := 'False'; ExternalVisible := 'False'; ExternalWritable := 'False'} : Bool;   // HMI Command - To Pos3
      H_CmdPos4 { ExternalAccessible := 'False'; ExternalVisible := 'False'; ExternalWritable := 'False'} : Bool;   // HMI Command - To Pos4
      H_CmdPos5 { ExternalAccessible := 'False'; ExternalVisible := 'False'; ExternalWritable := 'False'} : Bool;   // HMI Command - To Pos5
      H_CmdPosMaint { ExternalAccessible := 'False'; ExternalVisible := 'False'; ExternalWritable := 'False'} : Bool;   // HMI Command - To Maintenance Pos
   END_VAR
   VAR RETAIN
      H_ReferencingPos : DInt;   // Referencing position
   END_VAR
   VAR
      _SoftDetPos1 { ExternalAccessible := 'False'; ExternalVisible := 'False'; ExternalWritable := 'False'} : "LGBSoftDet";   // FB
      _SoftDetPos2 { ExternalAccessible := 'False'; ExternalVisible := 'False'; ExternalWritable := 'False'} : "LGBSoftDet";   // FB
      _SoftDetPos3 { ExternalAccessible := 'False'; ExternalVisible := 'False'; ExternalWritable := 'False'} : "LGBSoftDet";   // FB
      _SoftDetPos4 { ExternalAccessible := 'False'; ExternalVisible := 'False'; ExternalWritable := 'False'} : "LGBSoftDet";   // FB
      _SoftDetPos5 { ExternalAccessible := 'False'; ExternalVisible := 'False'; ExternalWritable := 'False'} : "LGBSoftDet";   // FB
      _SoftDetPosMaint { ExternalAccessible := 'False'; ExternalVisible := 'False'; ExternalWritable := 'False'} : "LGBSoftDet";   // FB
      _Motor { ExternalAccessible := 'False'; ExternalVisible := 'False'; ExternalWritable := 'False'} : "LGBMotor2W2S-MoviFitFCPN";   // FB
      _MovFunc2Pos2s { ExternalAccessible := 'False'; ExternalVisible := 'False'; ExternalWritable := 'False'} : "LMovFnc2Pos2S";   // FB
      _StopPos { ExternalAccessible := 'False'; ExternalVisible := 'False'; ExternalWritable := 'False'} : "L2StopPos";   // FB
      _OverTravelSet { ExternalAccessible := 'False'; ExternalVisible := 'False'; ExternalWritable := 'False'} : "L1AlarmMultiIn";   // FB
      _OverTravelRes { ExternalAccessible := 'False'; ExternalVisible := 'False'; ExternalWritable := 'False'} : "L1AlarmMultiIn";   // FB
      _HartingPlug400V { ExternalAccessible := 'False'; ExternalVisible := 'False'; ExternalWritable := 'False'} : "L1AlarmMultiIn";   // FB
      _HartingPlug24V { ExternalAccessible := 'False'; ExternalVisible := 'False'; ExternalWritable := 'False'} : "L1AlarmMultiIn";   // FB
      _KeepPositionPos1 { ExternalAccessible := 'False'; ExternalVisible := 'False'; ExternalWritable := 'False'} : "L1AlarmMultiIn";   // FB
      _KeepPositionPos2 { ExternalAccessible := 'False'; ExternalVisible := 'False'; ExternalWritable := 'False'} : "L1AlarmMultiIn";   // FB
      _KeepPositionPos3 { ExternalAccessible := 'False'; ExternalVisible := 'False'; ExternalWritable := 'False'} : "L1AlarmMultiIn";   // FB
      _KeepPositionPos4 { ExternalAccessible := 'False'; ExternalVisible := 'False'; ExternalWritable := 'False'} : "L1AlarmMultiIn";   // FB
      _KeepPositionPos5 { ExternalAccessible := 'False'; ExternalVisible := 'False'; ExternalWritable := 'False'} : "L1AlarmMultiIn";   // FB
      T_DelayPB { ExternalAccessible := 'False'; ExternalVisible := 'False'; ExternalWritable := 'False'} : TON_TIME;   // Timer
      Edge { ExternalAccessible := 'False'; ExternalVisible := 'False'; ExternalWritable := 'False'} : Array[0..20] of Bool;   // Flank
   END_VAR
   VAR_TEMP
      NotUsedH_HMI : "H_HMI";   // Animation
      H_HMIMotor : "H_HMI";   // Temp
      H_HMITemp : "H_HMI";   // Animation
      TempReal1 : Real;
      TempReal2 : Real;
      TempReal3 : Real;
   END_VAR
   VAR_TEMP   // added for the SCL form of the ladder/FBD networks
      _w1 : Bool;
      _w2 : Bool;
      _w3 : Bool;
      _w4 : Bool;
      _w5 : Bool;
   END_VAR
BEGIN

REGION Network 1: **** 1 - Inputs **** HMI Commands
   // Extract The Commands From HMI
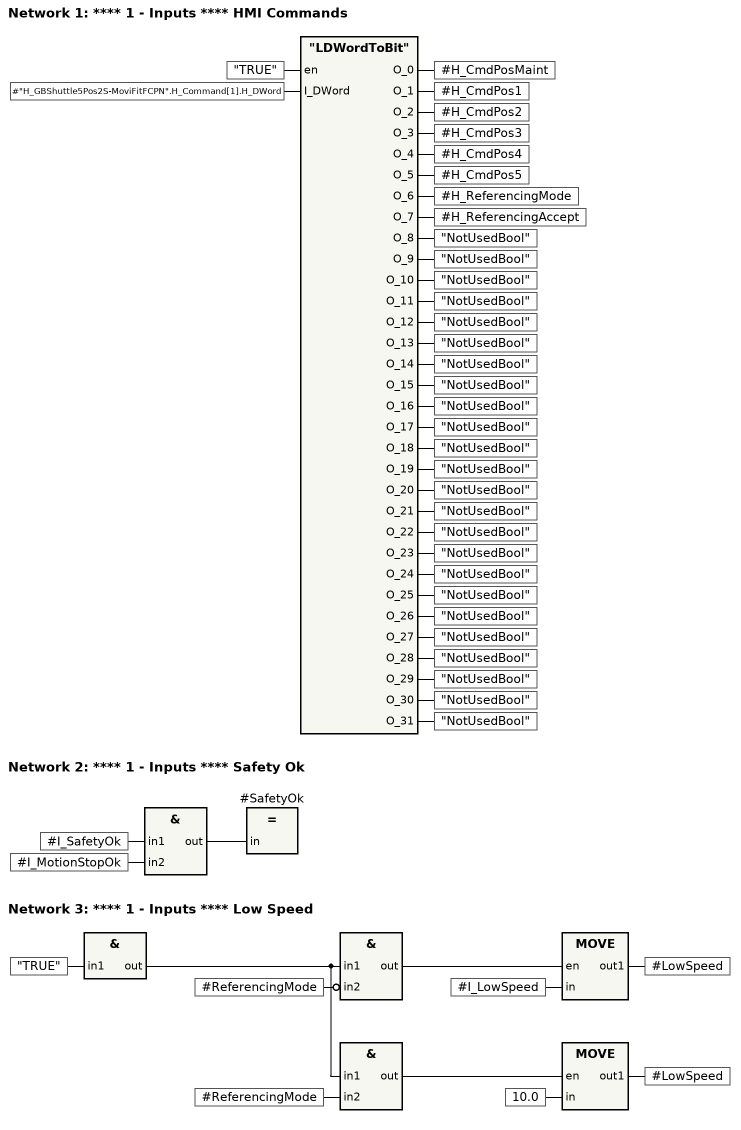
   IF "TRUE" THEN
       "LDWordToBit"(I_DWord := #"H_GBShuttle5Pos2S-MoviFitFCPN".H_Command[1].H_DWord,
                     O_0 => #H_CmdPosMaint,
                     O_1 => #H_CmdPos1,
                     O_2 => #H_CmdPos2,
                     O_3 => #H_CmdPos3,
                     O_4 => #H_CmdPos4,
                     O_5 => #H_CmdPos5,
                     O_6 => #H_ReferencingMode,
                     O_7 => #H_ReferencingAccept,
                     O_8 => "NotUsedBool",
                     O_9 => "NotUsedBool",
                     O_10 => "NotUsedBool",
                     O_11 => "NotUsedBool",
                     O_12 => "NotUsedBool",
                     O_13 => "NotUsedBool",
                     O_14 => "NotUsedBool",
                     O_15 => "NotUsedBool",
                     O_16 => "NotUsedBool",
                     O_17 => "NotUsedBool",
                     O_18 => "NotUsedBool",
                     O_19 => "NotUsedBool",
                     O_20 => "NotUsedBool",
                     O_21 => "NotUsedBool",
                     O_22 => "NotUsedBool",
                     O_23 => "NotUsedBool",
                     O_24 => "NotUsedBool",
                     O_25 => "NotUsedBool",
                     O_26 => "NotUsedBool",
                     O_27 => "NotUsedBool",
                     O_28 => "NotUsedBool",
                     O_29 => "NotUsedBool",
                     O_30 => "NotUsedBool",
                     O_31 => "NotUsedBool");
   END_IF;
END_REGION

REGION Network 2: **** 1 - Inputs **** Safety Ok
   #SafetyOk := #I_SafetyOk AND #I_MotionStopOk;
END_REGION

REGION Network 3: **** 1 - Inputs **** Low Speed
   IF "TRUE" AND NOT #ReferencingMode THEN #LowSpeed := #I_LowSpeed; END_IF;
   IF "TRUE" AND #ReferencingMode THEN #LowSpeed := 10.0; END_IF;
END_REGION

REGION Network 4: **** 1 - Inputs **** Lock local PB on position
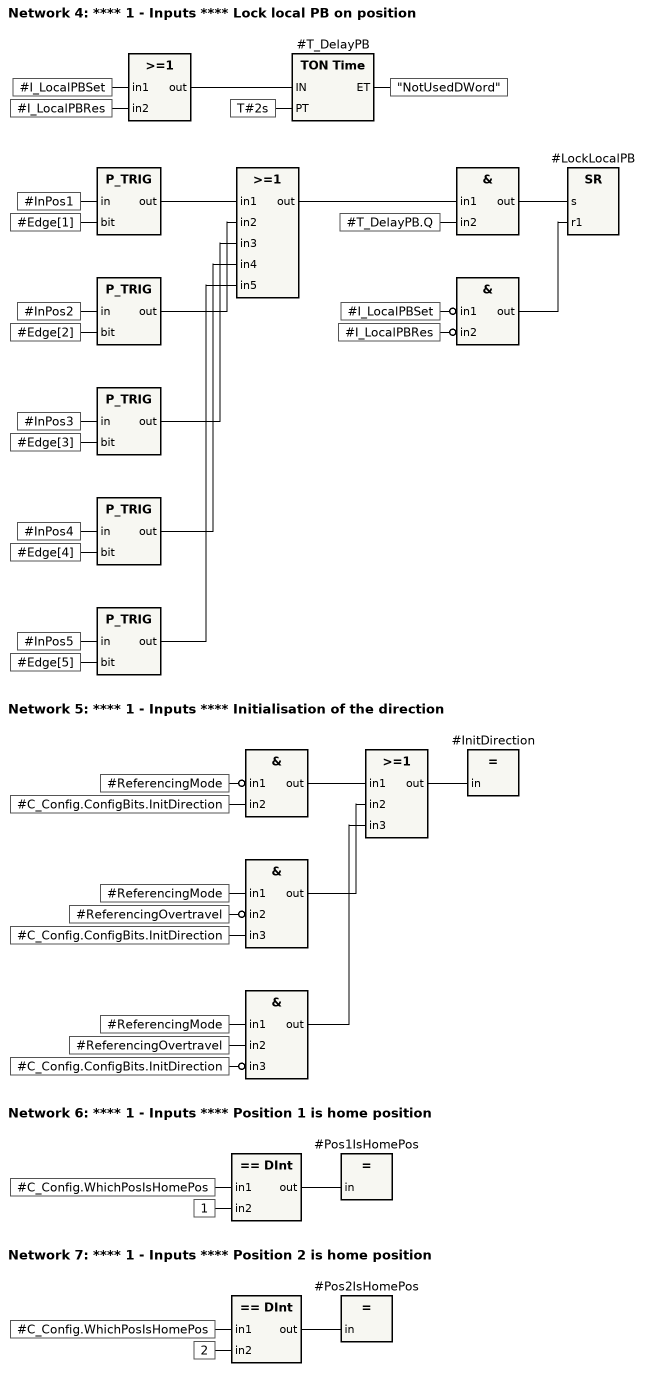
   #T_DelayPB(IN := #I_LocalPBSet OR #I_LocalPBRes, PT := T#2s, ET => "NotUsedDWord");   // TON
   #_w1 := #InPos1 AND NOT #Edge[1];   // rising edge
   #Edge[1] := #InPos1;
   #_w2 := #InPos2 AND NOT #Edge[2];   // rising edge
   #Edge[2] := #InPos2;
   #_w3 := #InPos3 AND NOT #Edge[3];   // rising edge
   #Edge[3] := #InPos3;
   #_w4 := #InPos4 AND NOT #Edge[4];   // rising edge
   #Edge[4] := #InPos4;
   #_w5 := #InPos5 AND NOT #Edge[5];   // rising edge
   #Edge[5] := #InPos5;
   IF (#_w1 OR #_w2 OR #_w3 OR #_w4 OR #_w5) AND #T_DelayPB.Q THEN
       #LockLocalPB := TRUE;   // SR flip-flop
   END_IF;
   IF NOT #I_LocalPBSet AND NOT #I_LocalPBRes THEN #LockLocalPB := FALSE; END_IF;
END_REGION

REGION Network 5: **** 1 - Inputs **** Initialisation of the direction
   #InitDirection := (NOT #ReferencingMode AND #C_Config.ConfigBits.InitDirection) OR (#ReferencingMode AND NOT #ReferencingOvertravel AND #C_Config.ConfigBits.InitDirection) OR (#ReferencingMode AND #ReferencingOvertravel AND NOT #C_Config.ConfigBits.InitDirection);
END_REGION

REGION Network 6: **** 1 - Inputs **** Position 1 is home position
   #Pos1IsHomePos := #C_Config.WhichPosIsHomePos = 1;
END_REGION

REGION Network 7: **** 1 - Inputs **** Position 2 is home position
   #Pos2IsHomePos := #C_Config.WhichPosIsHomePos = 2;
END_REGION

REGION Network 8: **** 1 - Inputs **** Position 3 is home position
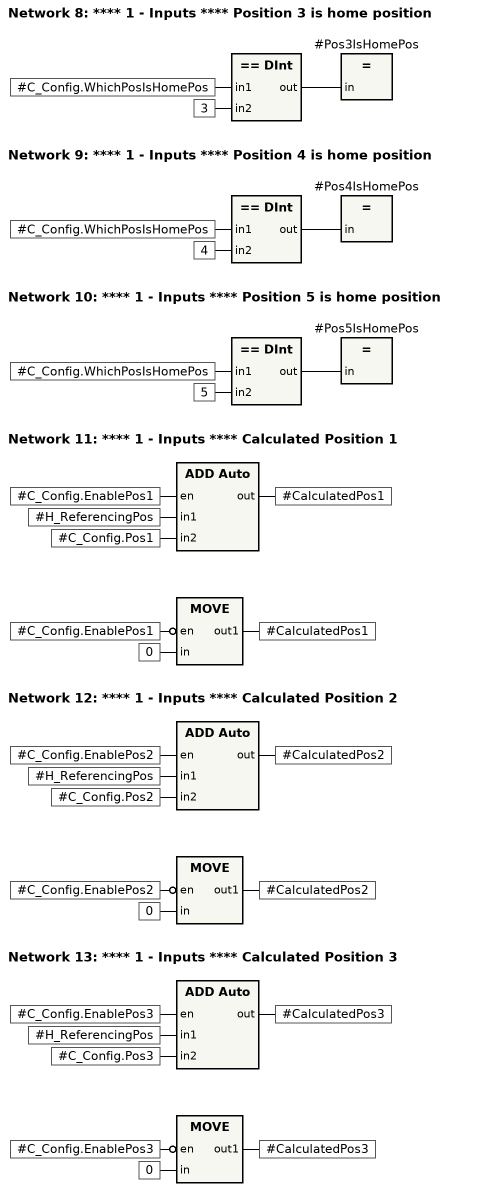
   #Pos3IsHomePos := #C_Config.WhichPosIsHomePos = 3;
END_REGION

REGION Network 9: **** 1 - Inputs **** Position 4 is home position
   #Pos4IsHomePos := #C_Config.WhichPosIsHomePos = 4;
END_REGION

REGION Network 10: **** 1 - Inputs **** Position 5 is home position
   #Pos5IsHomePos := #C_Config.WhichPosIsHomePos = 5;
END_REGION

REGION Network 11: **** 1 - Inputs **** Calculated Position 1
   IF #C_Config.EnablePos1 THEN #CalculatedPos1 := #H_ReferencingPos + #C_Config.Pos1; END_IF;
   IF NOT #C_Config.EnablePos1 THEN #CalculatedPos1 := 0; END_IF;
END_REGION

REGION Network 12: **** 1 - Inputs **** Calculated Position 2
   IF #C_Config.EnablePos2 THEN #CalculatedPos2 := #H_ReferencingPos + #C_Config.Pos2; END_IF;
   IF NOT #C_Config.EnablePos2 THEN #CalculatedPos2 := 0; END_IF;
END_REGION

REGION Network 13: **** 1 - Inputs **** Calculated Position 3
   IF #C_Config.EnablePos3 THEN #CalculatedPos3 := #H_ReferencingPos + #C_Config.Pos3; END_IF;
   IF NOT #C_Config.EnablePos3 THEN #CalculatedPos3 := 0; END_IF;
END_REGION

REGION Network 14: **** 1 - Inputs **** Calculated Position 4
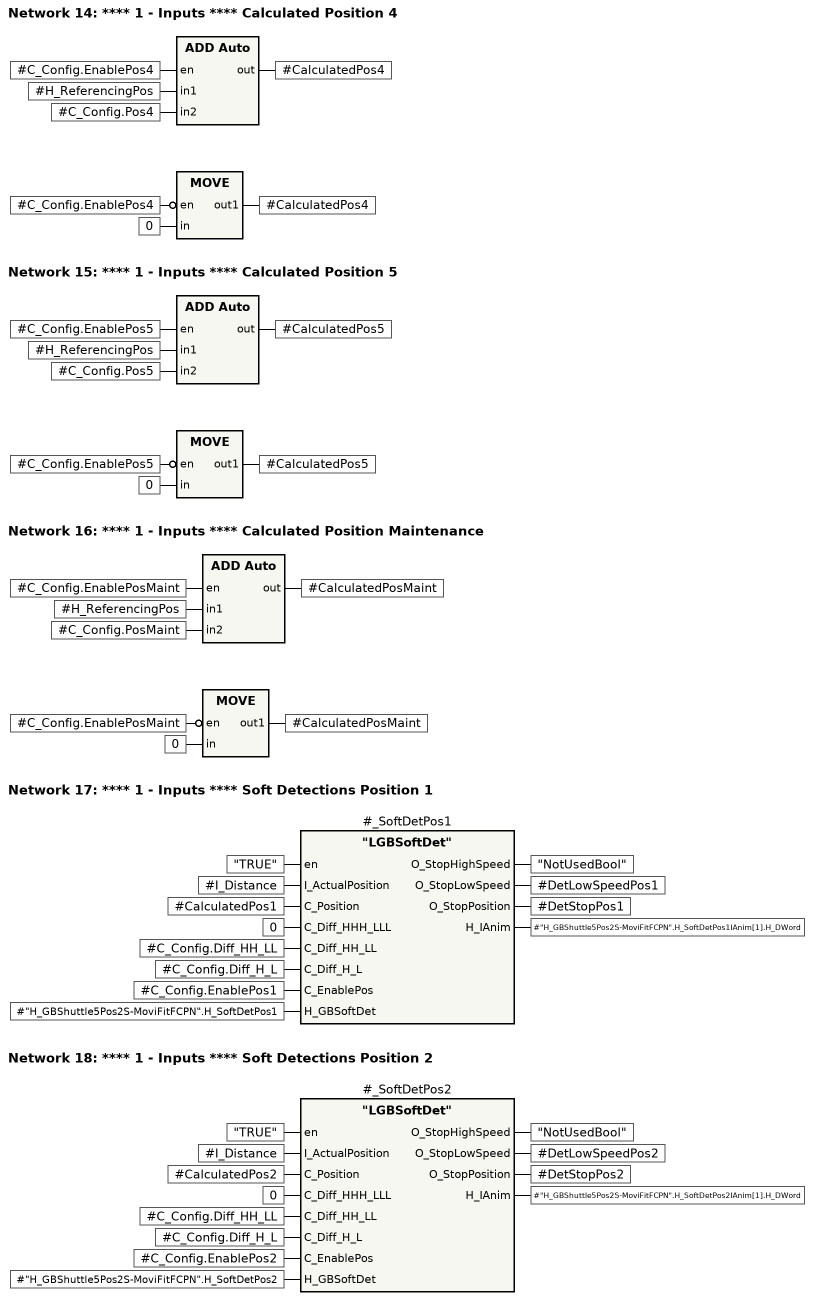
   IF #C_Config.EnablePos4 THEN #CalculatedPos4 := #H_ReferencingPos + #C_Config.Pos4; END_IF;
   IF NOT #C_Config.EnablePos4 THEN #CalculatedPos4 := 0; END_IF;
END_REGION

REGION Network 15: **** 1 - Inputs **** Calculated Position 5
   IF #C_Config.EnablePos5 THEN #CalculatedPos5 := #H_ReferencingPos + #C_Config.Pos5; END_IF;
   IF NOT #C_Config.EnablePos5 THEN #CalculatedPos5 := 0; END_IF;
END_REGION

REGION Network 16: **** 1 - Inputs **** Calculated Position Maintenance
   IF #C_Config.EnablePosMaint THEN #CalculatedPosMaint := #H_ReferencingPos + #C_Config.PosMaint; END_IF;
   IF NOT #C_Config.EnablePosMaint THEN #CalculatedPosMaint := 0; END_IF;
END_REGION

REGION Network 17: **** 1 - Inputs **** Soft Detections Position 1
   IF "TRUE" THEN
       #_SoftDetPos1(I_ActualPosition := #I_Distance,   // "LGBSoftDet"
                     C_Position := #CalculatedPos1,
                     C_Diff_HHH_LLL := 0,
                     C_Diff_HH_LL := #C_Config.Diff_HH_LL,
                     C_Diff_H_L := #C_Config.Diff_H_L,
                     C_EnablePos := #C_Config.EnablePos1,
                     H_GBSoftDet := #"H_GBShuttle5Pos2S-MoviFitFCPN".H_SoftDetPos1,
                     O_StopHighSpeed => "NotUsedBool",
                     O_StopLowSpeed => #DetLowSpeedPos1,
                     O_StopPosition => #DetStopPos1,
                     H_IAnim => #"H_GBShuttle5Pos2S-MoviFitFCPN".H_SoftDetPos1IAnim[1].H_DWord);
   END_IF;
END_REGION

REGION Network 18: **** 1 - Inputs **** Soft Detections Position 2
   IF "TRUE" THEN
       #_SoftDetPos2(I_ActualPosition := #I_Distance,   // "LGBSoftDet"
                     C_Position := #CalculatedPos2,
                     C_Diff_HHH_LLL := 0,
                     C_Diff_HH_LL := #C_Config.Diff_HH_LL,
                     C_Diff_H_L := #C_Config.Diff_H_L,
                     C_EnablePos := #C_Config.EnablePos2,
                     H_GBSoftDet := #"H_GBShuttle5Pos2S-MoviFitFCPN".H_SoftDetPos2,
                     O_StopHighSpeed => "NotUsedBool",
                     O_StopLowSpeed => #DetLowSpeedPos2,
                     O_StopPosition => #DetStopPos2,
                     H_IAnim => #"H_GBShuttle5Pos2S-MoviFitFCPN".H_SoftDetPos2IAnim[1].H_DWord);
   END_IF;
END_REGION

REGION Network 19: **** 1 - Inputs **** Soft Detections Position 3
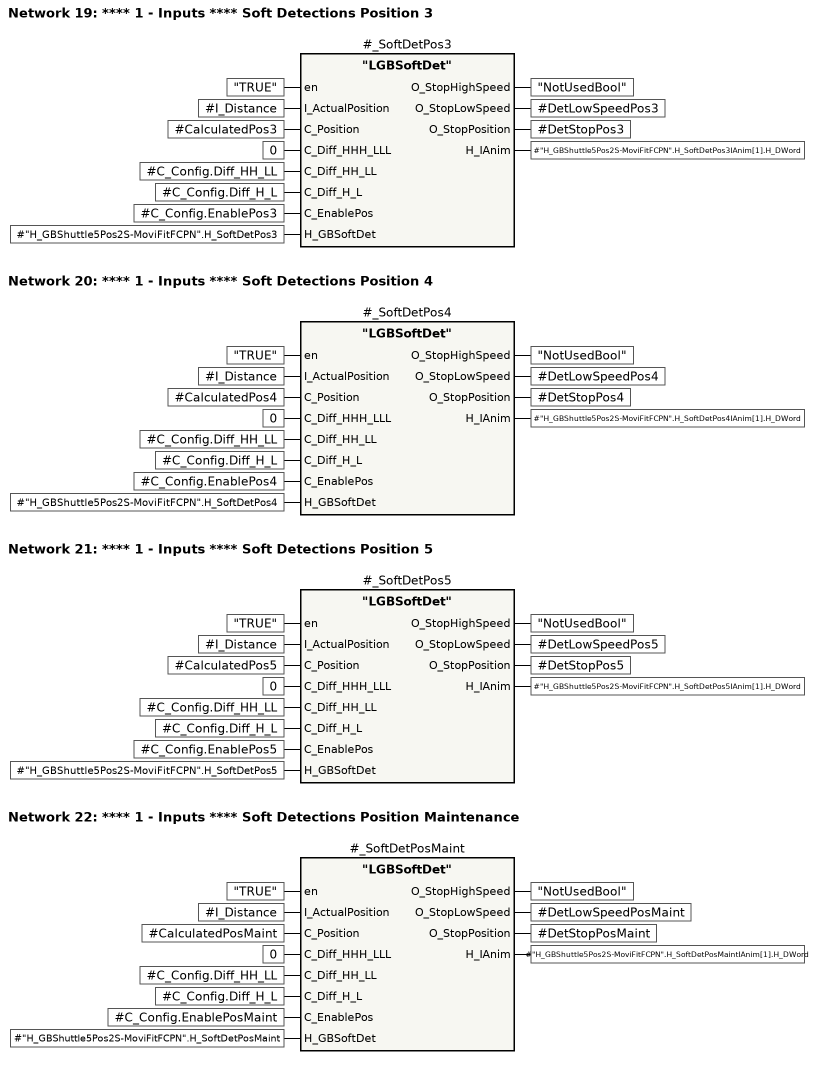
   IF "TRUE" THEN
       #_SoftDetPos3(I_ActualPosition := #I_Distance,   // "LGBSoftDet"
                     C_Position := #CalculatedPos3,
                     C_Diff_HHH_LLL := 0,
                     C_Diff_HH_LL := #C_Config.Diff_HH_LL,
                     C_Diff_H_L := #C_Config.Diff_H_L,
                     C_EnablePos := #C_Config.EnablePos3,
                     H_GBSoftDet := #"H_GBShuttle5Pos2S-MoviFitFCPN".H_SoftDetPos3,
                     O_StopHighSpeed => "NotUsedBool",
                     O_StopLowSpeed => #DetLowSpeedPos3,
                     O_StopPosition => #DetStopPos3,
                     H_IAnim => #"H_GBShuttle5Pos2S-MoviFitFCPN".H_SoftDetPos3IAnim[1].H_DWord);
   END_IF;
END_REGION

REGION Network 20: **** 1 - Inputs **** Soft Detections Position 4
   IF "TRUE" THEN
       #_SoftDetPos4(I_ActualPosition := #I_Distance,   // "LGBSoftDet"
                     C_Position := #CalculatedPos4,
                     C_Diff_HHH_LLL := 0,
                     C_Diff_HH_LL := #C_Config.Diff_HH_LL,
                     C_Diff_H_L := #C_Config.Diff_H_L,
                     C_EnablePos := #C_Config.EnablePos4,
                     H_GBSoftDet := #"H_GBShuttle5Pos2S-MoviFitFCPN".H_SoftDetPos4,
                     O_StopHighSpeed => "NotUsedBool",
                     O_StopLowSpeed => #DetLowSpeedPos4,
                     O_StopPosition => #DetStopPos4,
                     H_IAnim => #"H_GBShuttle5Pos2S-MoviFitFCPN".H_SoftDetPos4IAnim[1].H_DWord);
   END_IF;
END_REGION

REGION Network 21: **** 1 - Inputs **** Soft Detections Position 5
   IF "TRUE" THEN
       #_SoftDetPos5(I_ActualPosition := #I_Distance,   // "LGBSoftDet"
                     C_Position := #CalculatedPos5,
                     C_Diff_HHH_LLL := 0,
                     C_Diff_HH_LL := #C_Config.Diff_HH_LL,
                     C_Diff_H_L := #C_Config.Diff_H_L,
                     C_EnablePos := #C_Config.EnablePos5,
                     H_GBSoftDet := #"H_GBShuttle5Pos2S-MoviFitFCPN".H_SoftDetPos5,
                     O_StopHighSpeed => "NotUsedBool",
                     O_StopLowSpeed => #DetLowSpeedPos5,
                     O_StopPosition => #DetStopPos5,
                     H_IAnim => #"H_GBShuttle5Pos2S-MoviFitFCPN".H_SoftDetPos5IAnim[1].H_DWord);
   END_IF;
END_REGION

REGION Network 22: **** 1 - Inputs **** Soft Detections Position Maintenance
   IF "TRUE" THEN
       #_SoftDetPosMaint(I_ActualPosition := #I_Distance,   // "LGBSoftDet"
                         C_Position := #CalculatedPosMaint,
                         C_Diff_HHH_LLL := 0,
                         C_Diff_HH_LL := #C_Config.Diff_HH_LL,
                         C_Diff_H_L := #C_Config.Diff_H_L,
                         C_EnablePos := #C_Config.EnablePosMaint,
                         H_GBSoftDet := #"H_GBShuttle5Pos2S-MoviFitFCPN".H_SoftDetPosMaint,
                         O_StopHighSpeed => "NotUsedBool",
                         O_StopLowSpeed => #DetLowSpeedPosMaint,
                         O_StopPosition => #DetStopPosMaint,
                         H_IAnim => #"H_GBShuttle5Pos2S-MoviFitFCPN".H_SoftDetPosMaintIAnim[1].H_DWord);
   END_IF;
END_REGION

REGION Network 23: **** 1 - Inputs **** Direction Position 1
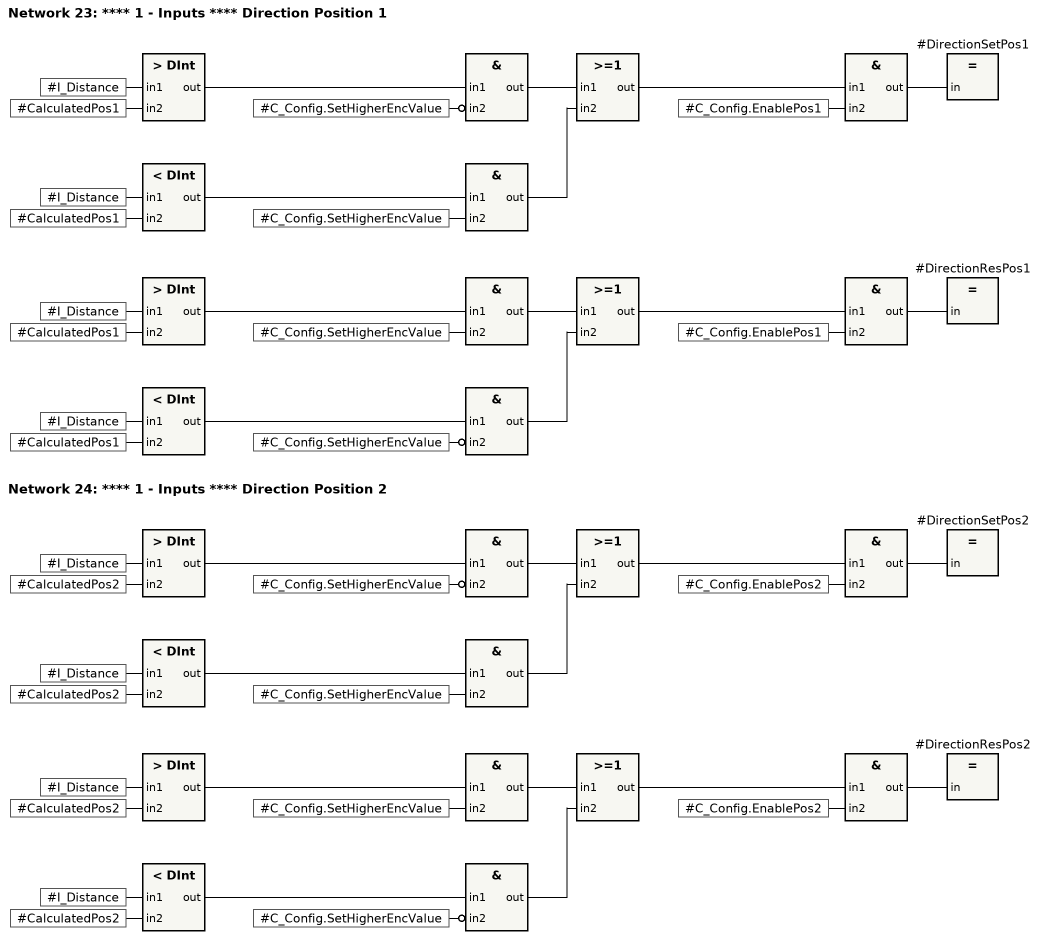
   #DirectionSetPos1 := (((#I_Distance > #CalculatedPos1) AND NOT #C_Config.SetHigherEncValue) OR ((#I_Distance < #CalculatedPos1) AND #C_Config.SetHigherEncValue)) AND #C_Config.EnablePos1;
   #DirectionResPos1 := (((#I_Distance > #CalculatedPos1) AND #C_Config.SetHigherEncValue) OR ((#I_Distance < #CalculatedPos1) AND NOT #C_Config.SetHigherEncValue)) AND #C_Config.EnablePos1;
END_REGION

REGION Network 24: **** 1 - Inputs **** Direction Position 2
   #DirectionSetPos2 := (((#I_Distance > #CalculatedPos2) AND NOT #C_Config.SetHigherEncValue) OR ((#I_Distance < #CalculatedPos2) AND #C_Config.SetHigherEncValue)) AND #C_Config.EnablePos2;
   #DirectionResPos2 := (((#I_Distance > #CalculatedPos2) AND #C_Config.SetHigherEncValue) OR ((#I_Distance < #CalculatedPos2) AND NOT #C_Config.SetHigherEncValue)) AND #C_Config.EnablePos2;
END_REGION

REGION Network 25: **** 1 - Inputs **** Direction Position 3
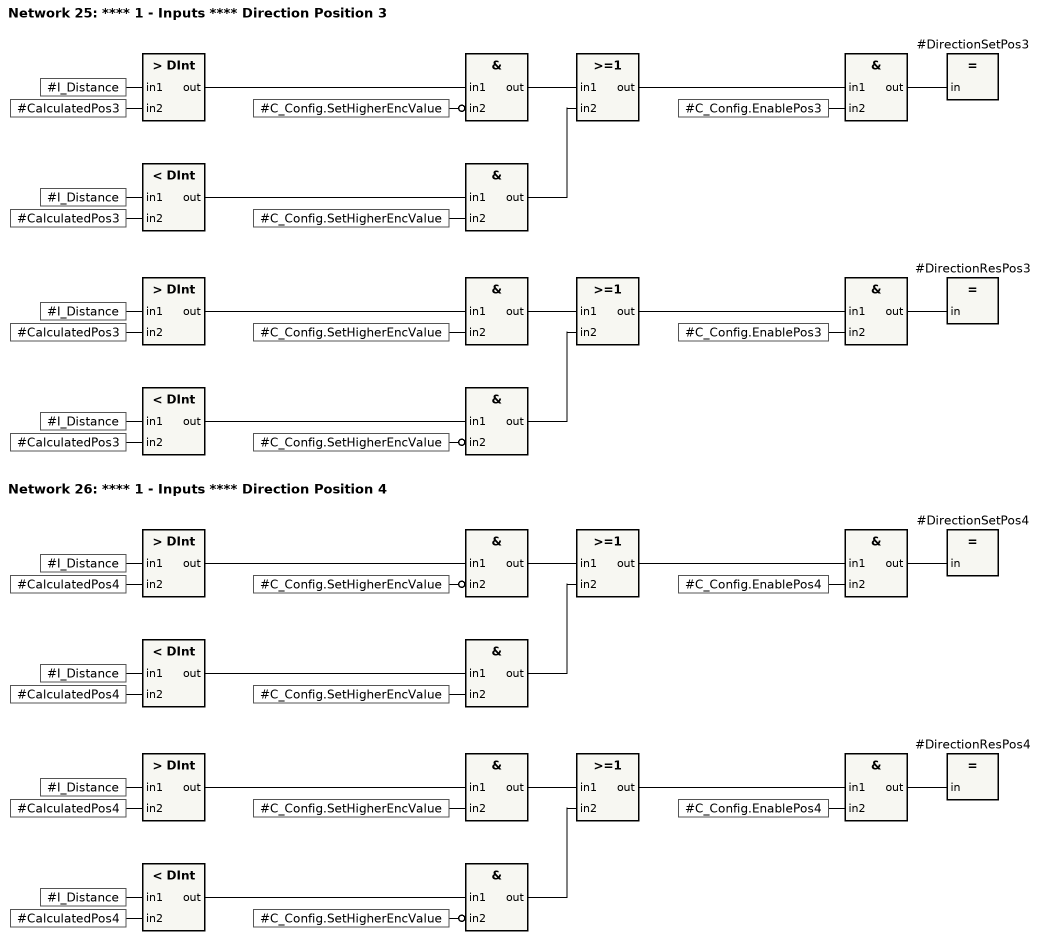
   #DirectionSetPos3 := (((#I_Distance > #CalculatedPos3) AND NOT #C_Config.SetHigherEncValue) OR ((#I_Distance < #CalculatedPos3) AND #C_Config.SetHigherEncValue)) AND #C_Config.EnablePos3;
   #DirectionResPos3 := (((#I_Distance > #CalculatedPos3) AND #C_Config.SetHigherEncValue) OR ((#I_Distance < #CalculatedPos3) AND NOT #C_Config.SetHigherEncValue)) AND #C_Config.EnablePos3;
END_REGION

REGION Network 26: **** 1 - Inputs **** Direction Position 4
   #DirectionSetPos4 := (((#I_Distance > #CalculatedPos4) AND NOT #C_Config.SetHigherEncValue) OR ((#I_Distance < #CalculatedPos4) AND #C_Config.SetHigherEncValue)) AND #C_Config.EnablePos4;
   #DirectionResPos4 := (((#I_Distance > #CalculatedPos4) AND #C_Config.SetHigherEncValue) OR ((#I_Distance < #CalculatedPos4) AND NOT #C_Config.SetHigherEncValue)) AND #C_Config.EnablePos4;
END_REGION

REGION Network 27: **** 1 - Inputs **** Direction Position 5
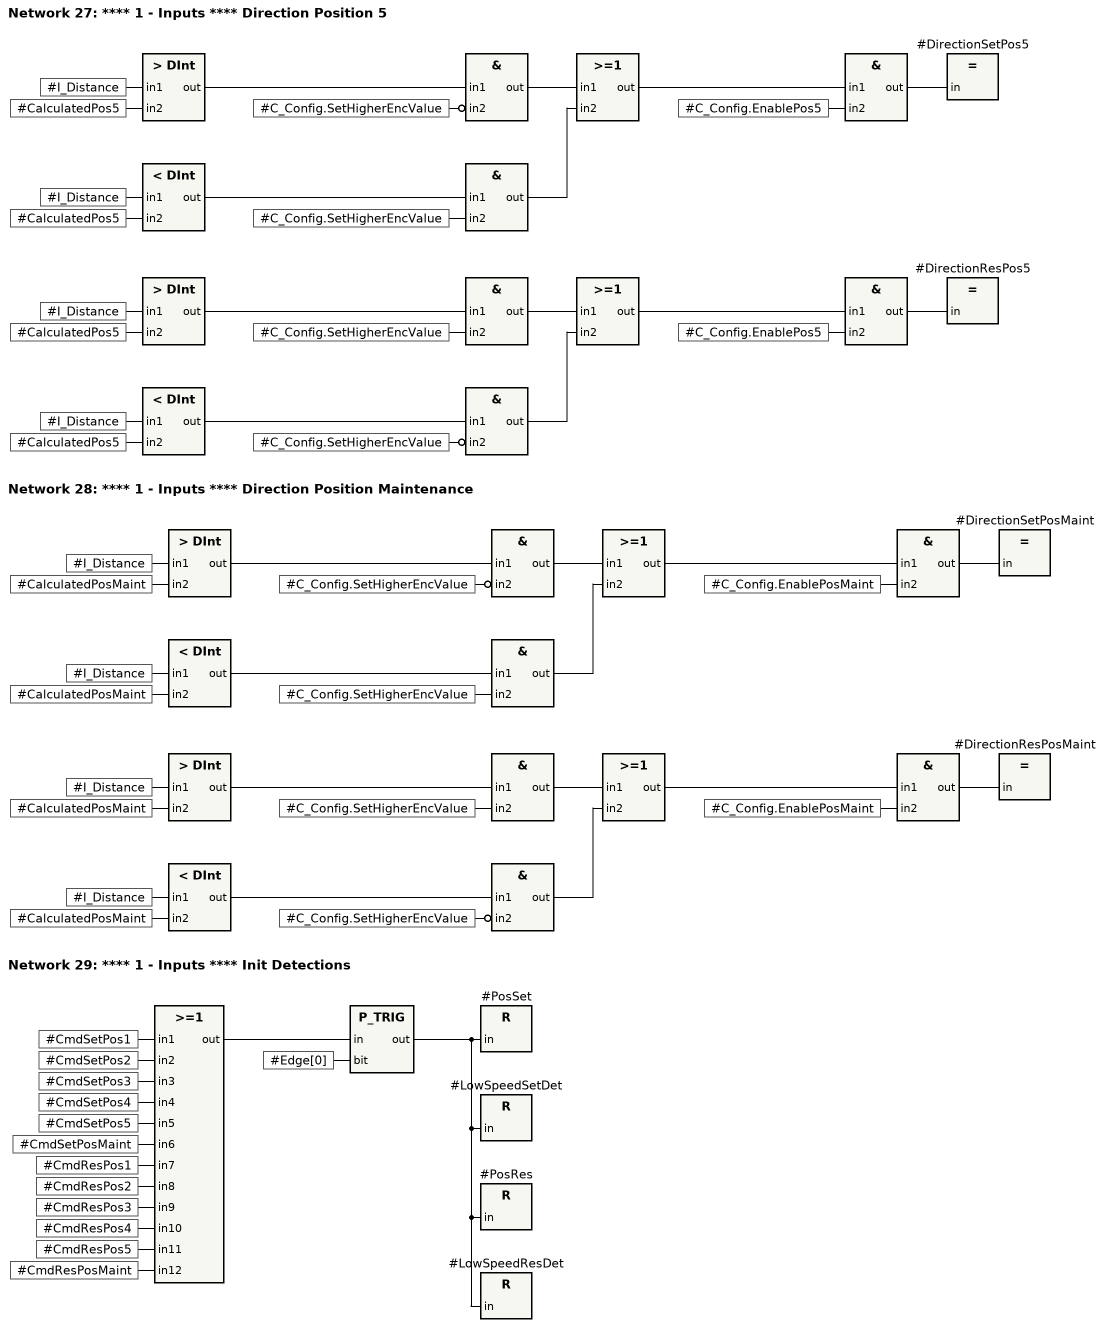
   #DirectionSetPos5 := (((#I_Distance > #CalculatedPos5) AND NOT #C_Config.SetHigherEncValue) OR ((#I_Distance < #CalculatedPos5) AND #C_Config.SetHigherEncValue)) AND #C_Config.EnablePos5;
   #DirectionResPos5 := (((#I_Distance > #CalculatedPos5) AND #C_Config.SetHigherEncValue) OR ((#I_Distance < #CalculatedPos5) AND NOT #C_Config.SetHigherEncValue)) AND #C_Config.EnablePos5;
END_REGION

REGION Network 28: **** 1 - Inputs **** Direction Position Maintenance
   #DirectionSetPosMaint := (((#I_Distance > #CalculatedPosMaint) AND NOT #C_Config.SetHigherEncValue) OR ((#I_Distance < #CalculatedPosMaint) AND #C_Config.SetHigherEncValue)) AND #C_Config.EnablePosMaint;
   #DirectionResPosMaint := (((#I_Distance > #CalculatedPosMaint) AND #C_Config.SetHigherEncValue) OR ((#I_Distance < #CalculatedPosMaint) AND NOT #C_Config.SetHigherEncValue)) AND #C_Config.EnablePosMaint;
END_REGION

REGION Network 29: **** 1 - Inputs **** Init Detections
   #_w1 := #CmdSetPos1 OR #CmdSetPos2 OR #CmdSetPos3 OR #CmdSetPos4 OR #CmdSetPos5 OR #CmdSetPosMaint OR #CmdResPos1 OR #CmdResPos2 OR #CmdResPos3 OR #CmdResPos4 OR #CmdResPos5 OR #CmdResPosMaint;
   #_w2 := #_w1 AND NOT #Edge[0];   // rising edge
   #Edge[0] := #_w1;
   IF #_w2 THEN
       #PosSet := FALSE;
       #LowSpeedSetDet := FALSE;
       #PosRes := FALSE;
       #LowSpeedResDet := FALSE;
   END_IF;
END_REGION

REGION Network 30: **** 1 - Inputs **** Detection -- Position Set
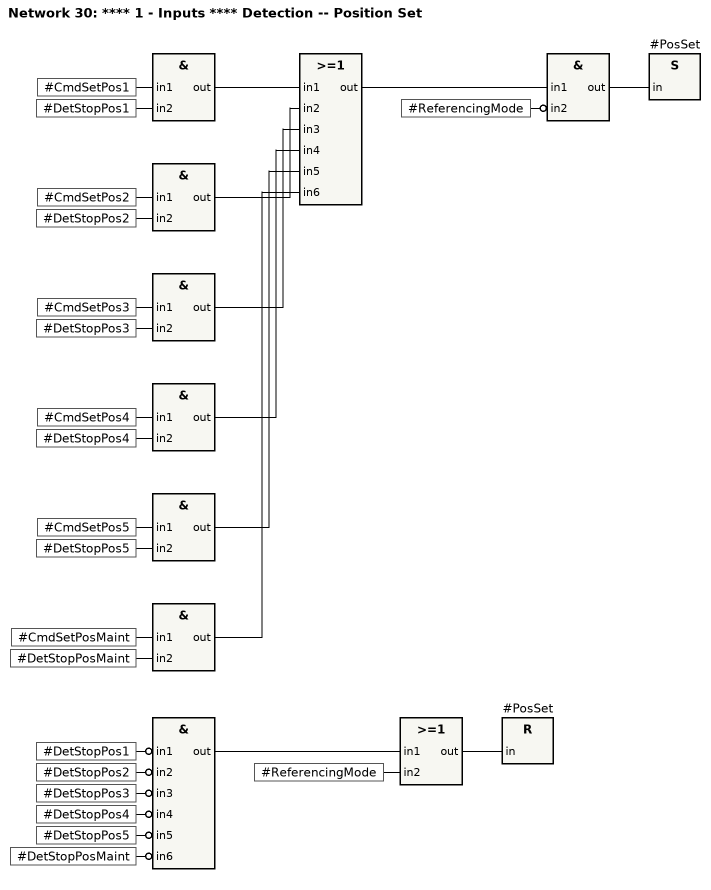
   IF ((#CmdSetPos1 AND #DetStopPos1) OR (#CmdSetPos2 AND #DetStopPos2) OR (#CmdSetPos3 AND #DetStopPos3) OR (#CmdSetPos4 AND #DetStopPos4) OR (#CmdSetPos5 AND #DetStopPos5) OR (#CmdSetPosMaint AND #DetStopPosMaint)) AND NOT #ReferencingMode THEN
       #PosSet := TRUE;
   END_IF;
   IF (NOT #DetStopPos1 AND NOT #DetStopPos2 AND NOT #DetStopPos3 AND NOT #DetStopPos4 AND NOT #DetStopPos5 AND NOT #DetStopPosMaint) OR #ReferencingMode THEN
       #PosSet := FALSE;
   END_IF;
END_REGION

REGION Network 31: **** 1 - Inputs **** Detection -- Position Set Slow
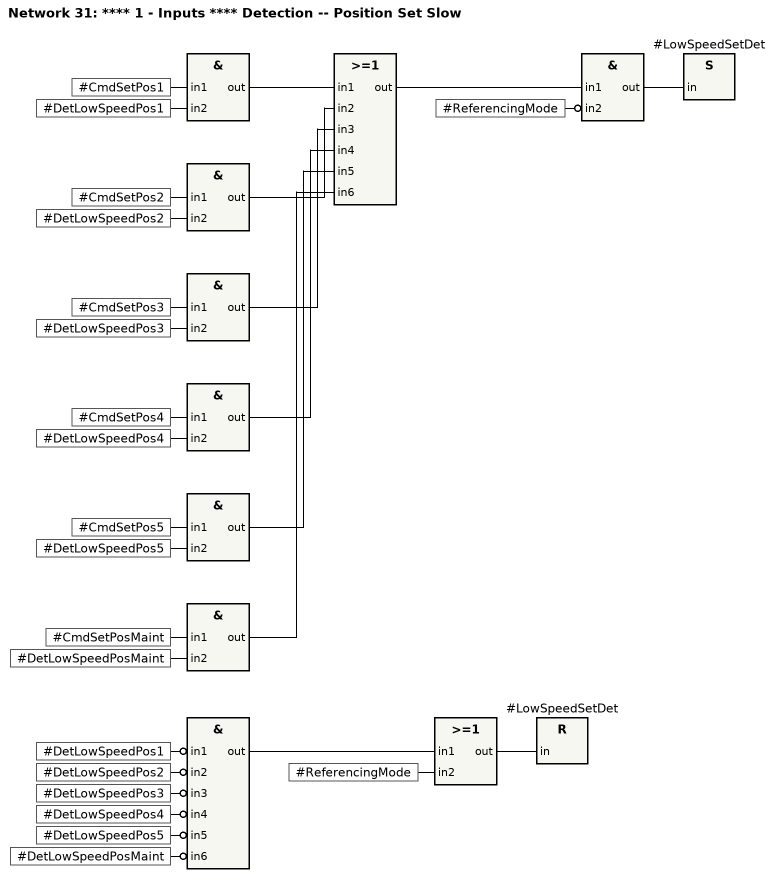
   IF ((#CmdSetPos1 AND #DetLowSpeedPos1) OR (#CmdSetPos2 AND #DetLowSpeedPos2) OR (#CmdSetPos3 AND #DetLowSpeedPos3) OR (#CmdSetPos4 AND #DetLowSpeedPos4) OR (#CmdSetPos5 AND #DetLowSpeedPos5) OR (#CmdSetPosMaint AND #DetLowSpeedPosMaint)) AND NOT #ReferencingMode THEN
       #LowSpeedSetDet := TRUE;
   END_IF;
   IF (NOT #DetLowSpeedPos1 AND NOT #DetLowSpeedPos2 AND NOT #DetLowSpeedPos3 AND NOT #DetLowSpeedPos4 AND NOT #DetLowSpeedPos5 AND NOT #DetLowSpeedPosMaint) OR #ReferencingMode THEN
       #LowSpeedSetDet := FALSE;
   END_IF;
END_REGION

REGION Network 32: **** 1 - Inputs **** Detection -- Position Reset
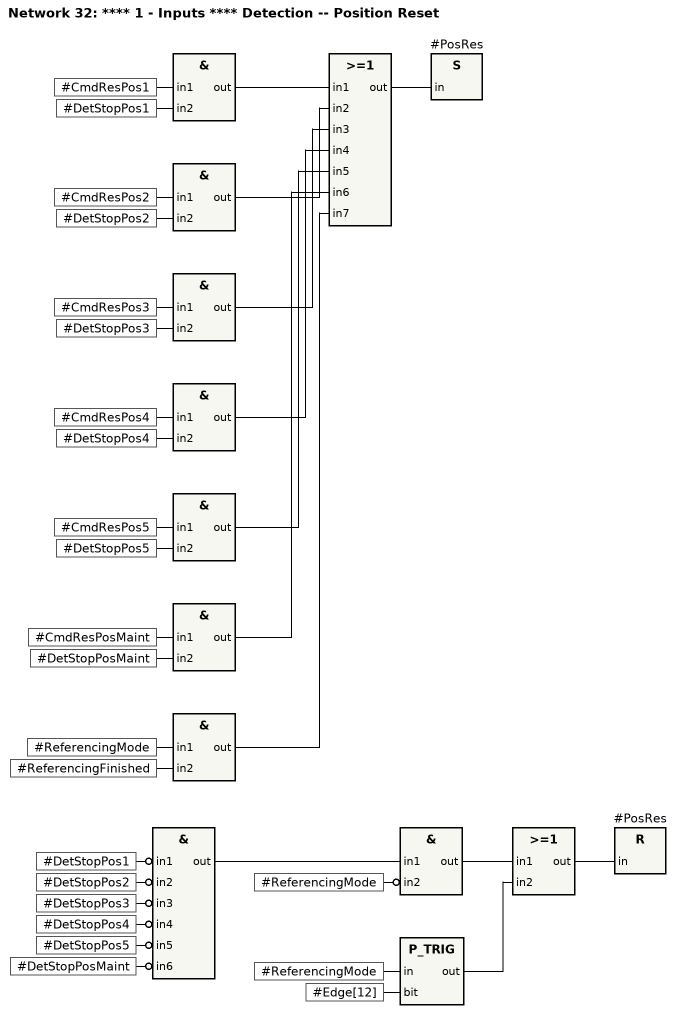
   IF (#CmdResPos1 AND #DetStopPos1) OR (#CmdResPos2 AND #DetStopPos2) OR (#CmdResPos3 AND #DetStopPos3) OR (#CmdResPos4 AND #DetStopPos4) OR (#CmdResPos5 AND #DetStopPos5) OR (#CmdResPosMaint AND #DetStopPosMaint) OR (#ReferencingMode AND #ReferencingFinished) THEN
       #PosRes := TRUE;
   END_IF;
   #_w1 := #ReferencingMode AND NOT #Edge[12];   // rising edge
   #Edge[12] := #ReferencingMode;
   IF (NOT #DetStopPos1 AND NOT #DetStopPos2 AND NOT #DetStopPos3 AND NOT #DetStopPos4 AND NOT #DetStopPos5 AND NOT #DetStopPosMaint AND NOT #ReferencingMode) OR #_w1 THEN
       #PosRes := FALSE;
   END_IF;
END_REGION

REGION Network 33: **** 1 - Inputs **** Detection -- Position Reset Slow
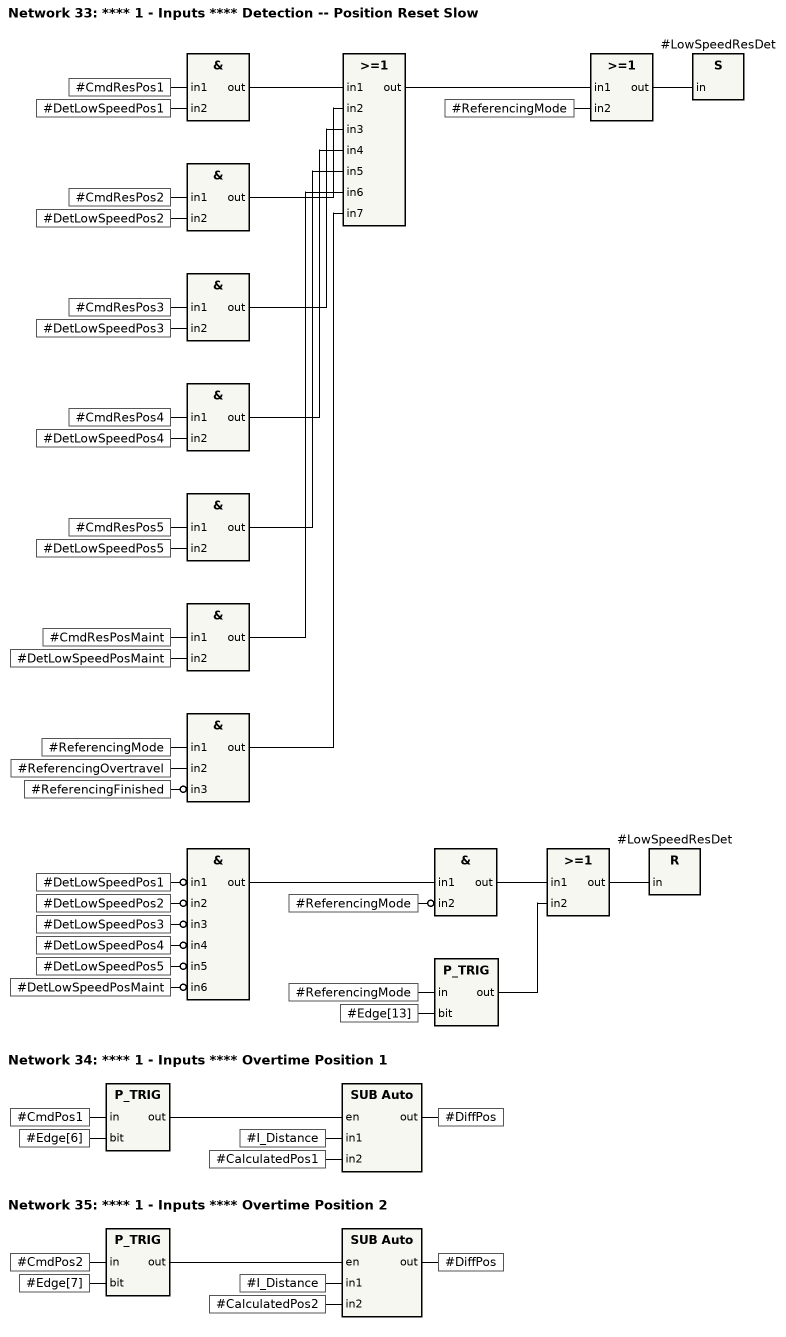
   IF (#CmdResPos1 AND #DetLowSpeedPos1) OR (#CmdResPos2 AND #DetLowSpeedPos2) OR (#CmdResPos3 AND #DetLowSpeedPos3) OR (#CmdResPos4 AND #DetLowSpeedPos4) OR (#CmdResPos5 AND #DetLowSpeedPos5) OR (#CmdResPosMaint AND #DetLowSpeedPosMaint) OR (#ReferencingMode AND #ReferencingOvertravel AND NOT #ReferencingFinished) OR #ReferencingMode THEN
       #LowSpeedResDet := TRUE;
   END_IF;
   #_w1 := #ReferencingMode AND NOT #Edge[13];   // rising edge
   #Edge[13] := #ReferencingMode;
   IF (NOT #DetLowSpeedPos1 AND NOT #DetLowSpeedPos2 AND NOT #DetLowSpeedPos3 AND NOT #DetLowSpeedPos4 AND NOT #DetLowSpeedPos5 AND NOT #DetLowSpeedPosMaint AND NOT #ReferencingMode) OR #_w1 THEN
       #LowSpeedResDet := FALSE;
   END_IF;
END_REGION

REGION Network 34: **** 1 - Inputs **** Overtime Position 1
   #_w1 := #CmdPos1 AND NOT #Edge[6];   // rising edge
   #Edge[6] := #CmdPos1;
   IF #_w1 THEN #DiffPos := #I_Distance - #CalculatedPos1; END_IF;
END_REGION

REGION Network 35: **** 1 - Inputs **** Overtime Position 2
   #_w1 := #CmdPos2 AND NOT #Edge[7];   // rising edge
   #Edge[7] := #CmdPos2;
   IF #_w1 THEN #DiffPos := #I_Distance - #CalculatedPos2; END_IF;
END_REGION

REGION Network 36: **** 1 - Inputs **** Overtime Position 3
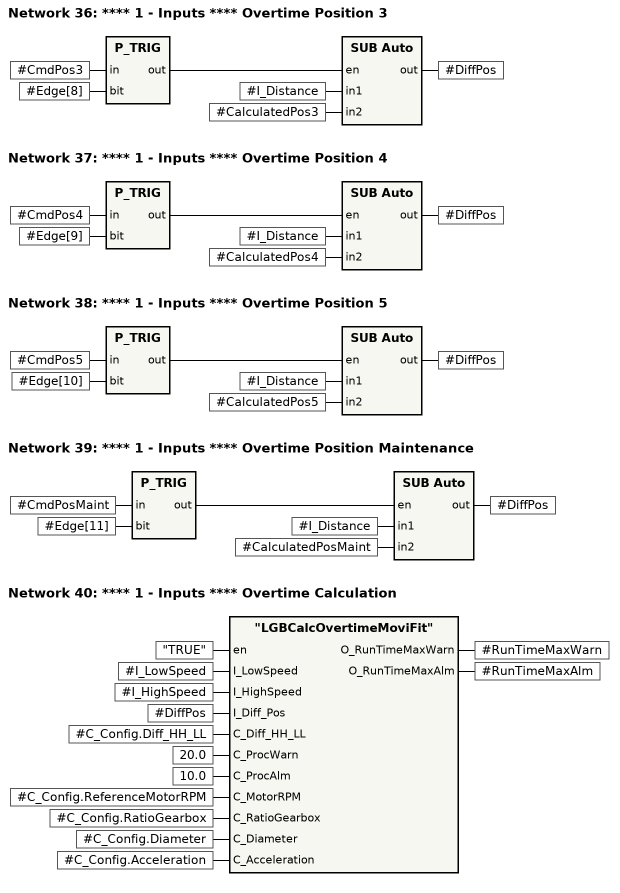
   #_w1 := #CmdPos3 AND NOT #Edge[8];   // rising edge
   #Edge[8] := #CmdPos3;
   IF #_w1 THEN #DiffPos := #I_Distance - #CalculatedPos3; END_IF;
END_REGION

REGION Network 37: **** 1 - Inputs **** Overtime Position 4
   #_w1 := #CmdPos4 AND NOT #Edge[9];   // rising edge
   #Edge[9] := #CmdPos4;
   IF #_w1 THEN #DiffPos := #I_Distance - #CalculatedPos4; END_IF;
END_REGION

REGION Network 38: **** 1 - Inputs **** Overtime Position 5
   #_w1 := #CmdPos5 AND NOT #Edge[10];   // rising edge
   #Edge[10] := #CmdPos5;
   IF #_w1 THEN #DiffPos := #I_Distance - #CalculatedPos5; END_IF;
END_REGION

REGION Network 39: **** 1 - Inputs **** Overtime Position Maintenance
   #_w1 := #CmdPosMaint AND NOT #Edge[11];   // rising edge
   #Edge[11] := #CmdPosMaint;
   IF #_w1 THEN #DiffPos := #I_Distance - #CalculatedPosMaint; END_IF;
END_REGION

REGION Network 40: **** 1 - Inputs **** Overtime Calculation
   IF "TRUE" THEN
       "LGBCalcOvertimeMoviFit"(I_LowSpeed := #I_LowSpeed,
                               I_HighSpeed := #I_HighSpeed,
                               I_Diff_Pos := #DiffPos,
                               C_Diff_HH_LL := #C_Config.Diff_HH_LL,
                               C_ProcWarn := 20.0,
                               C_ProcAlm := 10.0,
                               C_MotorRPM := #C_Config.ReferenceMotorRPM,
                               C_RatioGearbox := #C_Config.RatioGearbox,
                               C_Diameter := #C_Config.Diameter,
                               C_Acceleration := #C_Config.Acceleration,
                               O_RunTimeMaxWarn => #RunTimeMaxWarn,
                               O_RunTimeMaxAlm => #RunTimeMaxAlm);
   END_IF;
END_REGION

REGION Network 41: **** 1 - Inputs **** Overtime Result
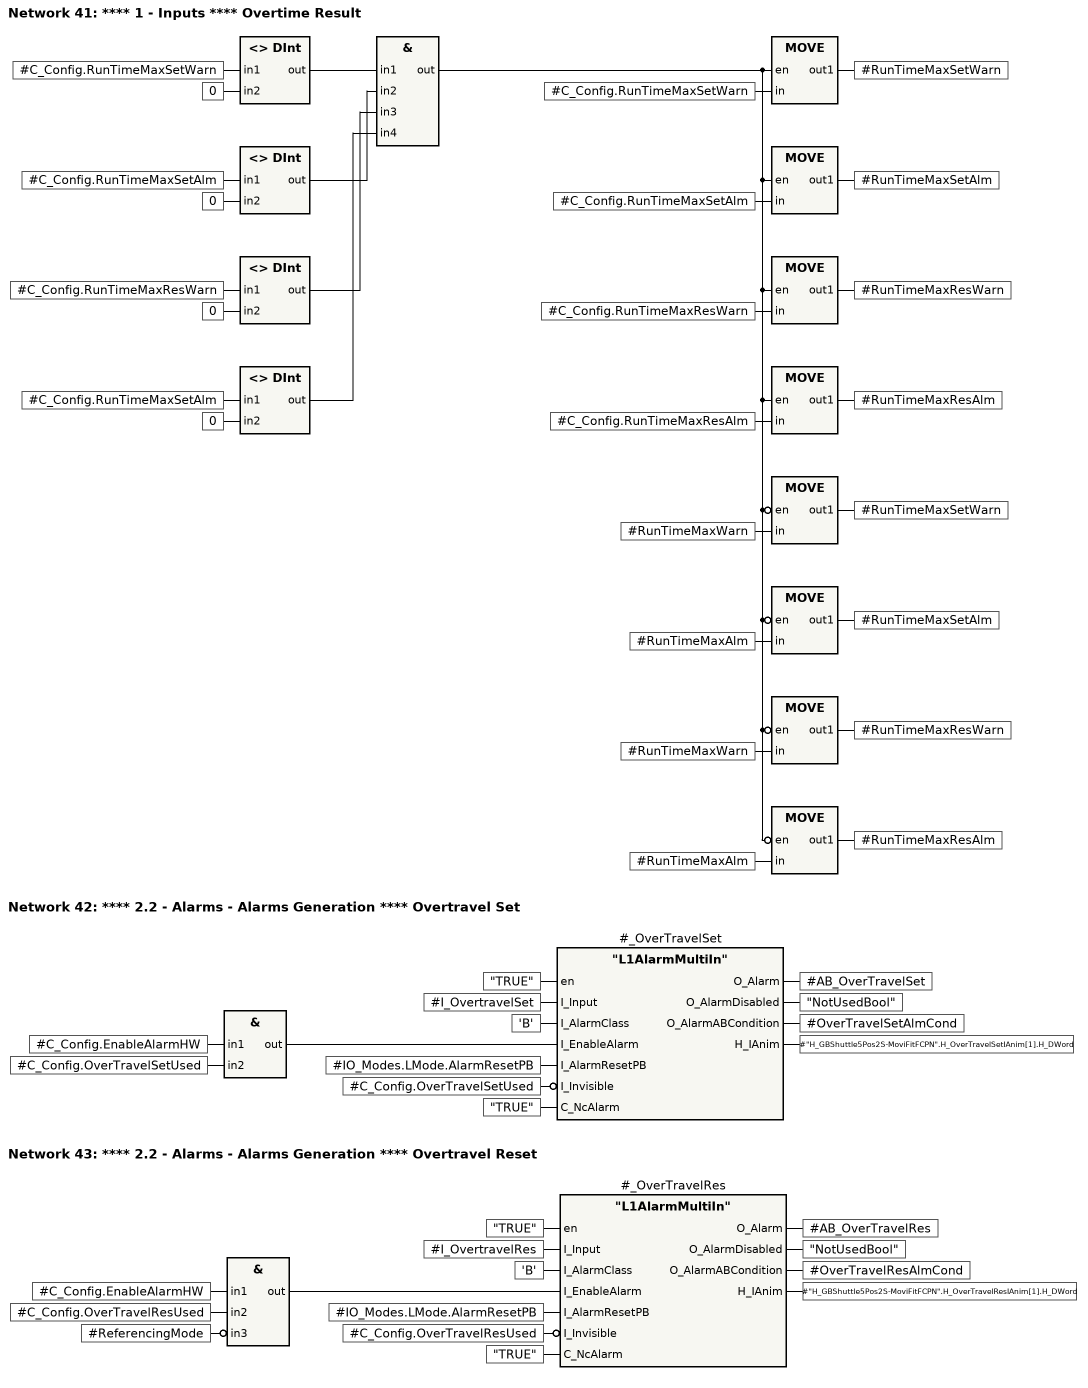
   #_w1 := (#C_Config.RunTimeMaxSetWarn <> 0) AND (#C_Config.RunTimeMaxSetAlm <> 0) AND (#C_Config.RunTimeMaxResWarn <> 0) AND (#C_Config.RunTimeMaxSetAlm <> 0);
   IF #_w1 THEN
       #RunTimeMaxSetWarn := #C_Config.RunTimeMaxSetWarn;
       #RunTimeMaxSetAlm := #C_Config.RunTimeMaxSetAlm;
       #RunTimeMaxResWarn := #C_Config.RunTimeMaxResWarn;
       #RunTimeMaxResAlm := #C_Config.RunTimeMaxResAlm;
   END_IF;
   IF NOT #_w1 THEN
       #RunTimeMaxSetWarn := #RunTimeMaxWarn;
       #RunTimeMaxSetAlm := #RunTimeMaxAlm;
       #RunTimeMaxResWarn := #RunTimeMaxWarn;
       #RunTimeMaxResAlm := #RunTimeMaxAlm;
   END_IF;
END_REGION

REGION Network 42: **** 2.2 - Alarms - Alarms Generation **** Overtravel Set
   IF "TRUE" THEN
       #_OverTravelSet(I_Input := #I_OvertravelSet,   // "L1AlarmMultiIn"
                       I_AlarmClass := 'B',
                       I_EnableAlarm := #C_Config.EnableAlarmHW AND #C_Config.OverTravelSetUsed,
                       I_AlarmResetPB := #IO_Modes.LMode.AlarmResetPB,
                       I_Invisible := NOT #C_Config.OverTravelSetUsed,
                       C_NcAlarm := "TRUE",
                       O_Alarm => #AB_OverTravelSet,
                       O_AlarmDisabled => "NotUsedBool",
                       O_AlarmABCondition => #OverTravelSetAlmCond,
                       H_IAnim => #"H_GBShuttle5Pos2S-MoviFitFCPN".H_OverTravelSetIAnim[1].H_DWord);
   END_IF;
END_REGION

REGION Network 43: **** 2.2 - Alarms - Alarms Generation **** Overtravel Reset
   IF "TRUE" THEN
       #_OverTravelRes(I_Input := #I_OvertravelRes,   // "L1AlarmMultiIn"
                       I_AlarmClass := 'B',
                       I_EnableAlarm := #C_Config.EnableAlarmHW AND #C_Config.OverTravelResUsed AND NOT #ReferencingMode,
                       I_AlarmResetPB := #IO_Modes.LMode.AlarmResetPB,
                       I_Invisible := NOT #C_Config.OverTravelResUsed,
                       C_NcAlarm := "TRUE",
                       O_Alarm => #AB_OverTravelRes,
                       O_AlarmDisabled => "NotUsedBool",
                       O_AlarmABCondition => #OverTravelResAlmCond,
                       H_IAnim => #"H_GBShuttle5Pos2S-MoviFitFCPN".H_OverTravelResIAnim[1].H_DWord);
   END_IF;
END_REGION

REGION Network 44: **** 2.2 - Alarms - Alarms Generation **** Harting plug 400VAC
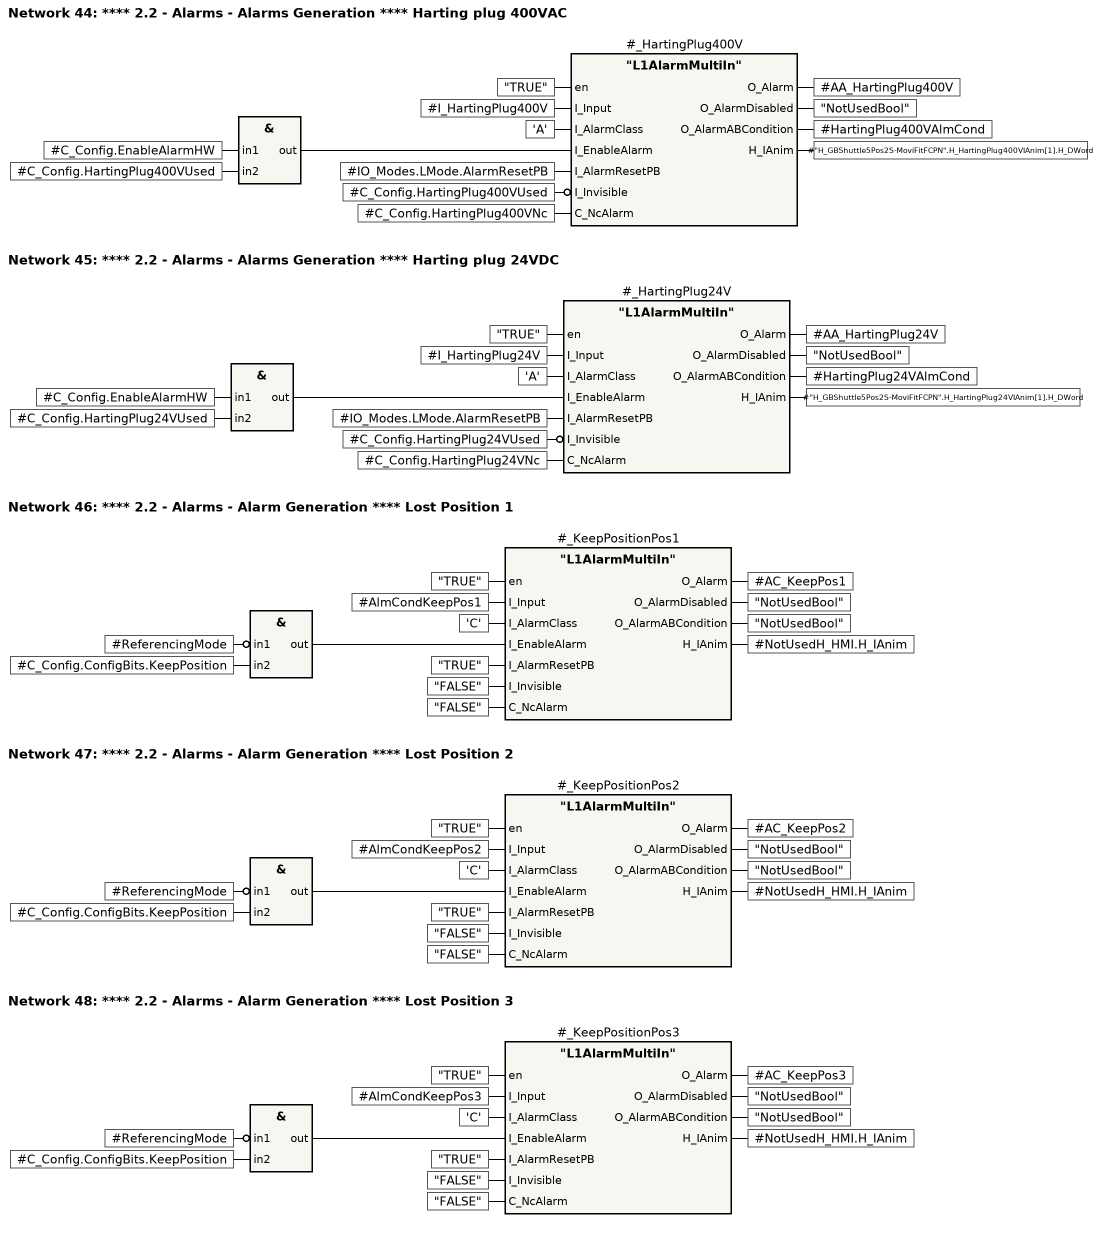
   IF "TRUE" THEN
       #_HartingPlug400V(I_Input := #I_HartingPlug400V,   // "L1AlarmMultiIn"
                         I_AlarmClass := 'A',
                         I_EnableAlarm := #C_Config.EnableAlarmHW AND #C_Config.HartingPlug400VUsed,
                         I_AlarmResetPB := #IO_Modes.LMode.AlarmResetPB,
                         I_Invisible := NOT #C_Config.HartingPlug400VUsed,
                         C_NcAlarm := #C_Config.HartingPlug400VNc,
                         O_Alarm => #AA_HartingPlug400V,
                         O_AlarmDisabled => "NotUsedBool",
                         O_AlarmABCondition => #HartingPlug400VAlmCond,
                         H_IAnim => #"H_GBShuttle5Pos2S-MoviFitFCPN".H_HartingPlug400VIAnim[1].H_DWord);
   END_IF;
END_REGION

REGION Network 45: **** 2.2 - Alarms - Alarms Generation **** Harting plug 24VDC
   IF "TRUE" THEN
       #_HartingPlug24V(I_Input := #I_HartingPlug24V,   // "L1AlarmMultiIn"
                        I_AlarmClass := 'A',
                        I_EnableAlarm := #C_Config.EnableAlarmHW AND #C_Config.HartingPlug24VUsed,
                        I_AlarmResetPB := #IO_Modes.LMode.AlarmResetPB,
                        I_Invisible := NOT #C_Config.HartingPlug24VUsed,
                        C_NcAlarm := #C_Config.HartingPlug24VNc,
                        O_Alarm => #AA_HartingPlug24V,
                        O_AlarmDisabled => "NotUsedBool",
                        O_AlarmABCondition => #HartingPlug24VAlmCond,
                        H_IAnim => #"H_GBShuttle5Pos2S-MoviFitFCPN".H_HartingPlug24VIAnim[1].H_DWord);
   END_IF;
END_REGION

REGION Network 46: **** 2.2 - Alarms - Alarm Generation **** Lost Position 1
   IF "TRUE" THEN
       #_KeepPositionPos1(I_Input := #AlmCondKeepPos1,   // "L1AlarmMultiIn"
                          I_AlarmClass := 'C',
                          I_EnableAlarm := NOT #ReferencingMode AND #C_Config.ConfigBits.KeepPosition,
                          I_AlarmResetPB := "TRUE",
                          I_Invisible := "FALSE",
                          C_NcAlarm := "FALSE",
                          O_Alarm => #AC_KeepPos1,
                          O_AlarmDisabled => "NotUsedBool",
                          O_AlarmABCondition => "NotUsedBool",
                          H_IAnim => #NotUsedH_HMI.H_IAnim);
   END_IF;
END_REGION

REGION Network 47: **** 2.2 - Alarms - Alarm Generation **** Lost Position 2
   IF "TRUE" THEN
       #_KeepPositionPos2(I_Input := #AlmCondKeepPos2,   // "L1AlarmMultiIn"
                          I_AlarmClass := 'C',
                          I_EnableAlarm := NOT #ReferencingMode AND #C_Config.ConfigBits.KeepPosition,
                          I_AlarmResetPB := "TRUE",
                          I_Invisible := "FALSE",
                          C_NcAlarm := "FALSE",
                          O_Alarm => #AC_KeepPos2,
                          O_AlarmDisabled => "NotUsedBool",
                          O_AlarmABCondition => "NotUsedBool",
                          H_IAnim => #NotUsedH_HMI.H_IAnim);
   END_IF;
END_REGION

REGION Network 48: **** 2.2 - Alarms - Alarm Generation **** Lost Position 3
   IF "TRUE" THEN
       #_KeepPositionPos3(I_Input := #AlmCondKeepPos3,   // "L1AlarmMultiIn"
                          I_AlarmClass := 'C',
                          I_EnableAlarm := NOT #ReferencingMode AND #C_Config.ConfigBits.KeepPosition,
                          I_AlarmResetPB := "TRUE",
                          I_Invisible := "FALSE",
                          C_NcAlarm := "FALSE",
                          O_Alarm => #AC_KeepPos3,
                          O_AlarmDisabled => "NotUsedBool",
                          O_AlarmABCondition => "NotUsedBool",
                          H_IAnim => #NotUsedH_HMI.H_IAnim);
   END_IF;
END_REGION

REGION Network 49: **** 2.2 - Alarms - Alarm Generation **** Lost Position 4
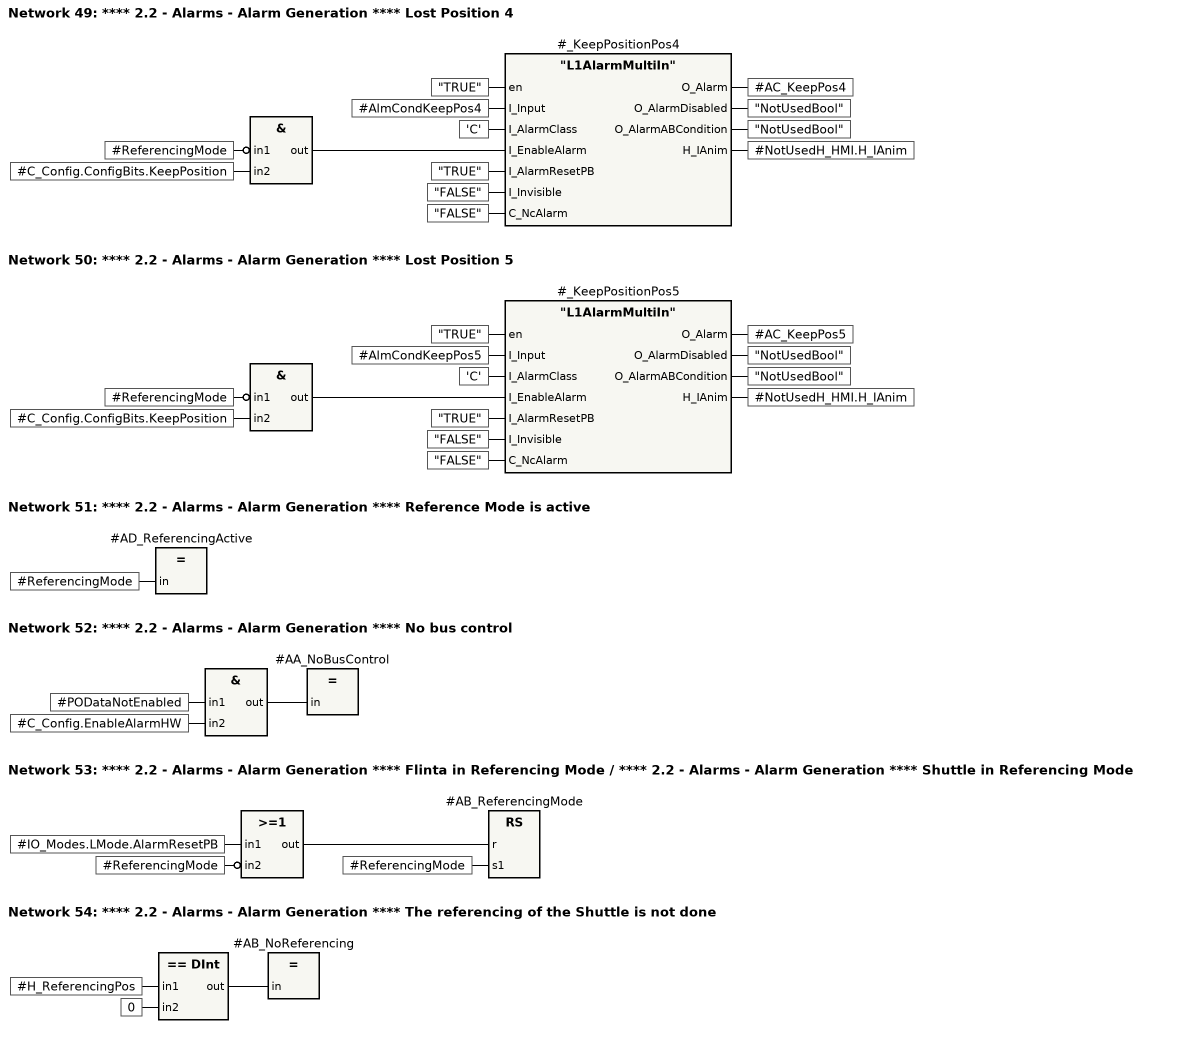
   IF "TRUE" THEN
       #_KeepPositionPos4(I_Input := #AlmCondKeepPos4,   // "L1AlarmMultiIn"
                          I_AlarmClass := 'C',
                          I_EnableAlarm := NOT #ReferencingMode AND #C_Config.ConfigBits.KeepPosition,
                          I_AlarmResetPB := "TRUE",
                          I_Invisible := "FALSE",
                          C_NcAlarm := "FALSE",
                          O_Alarm => #AC_KeepPos4,
                          O_AlarmDisabled => "NotUsedBool",
                          O_AlarmABCondition => "NotUsedBool",
                          H_IAnim => #NotUsedH_HMI.H_IAnim);
   END_IF;
END_REGION

REGION Network 50: **** 2.2 - Alarms - Alarm Generation **** Lost Position 5
   IF "TRUE" THEN
       #_KeepPositionPos5(I_Input := #AlmCondKeepPos5,   // "L1AlarmMultiIn"
                          I_AlarmClass := 'C',
                          I_EnableAlarm := NOT #ReferencingMode AND #C_Config.ConfigBits.KeepPosition,
                          I_AlarmResetPB := "TRUE",
                          I_Invisible := "FALSE",
                          C_NcAlarm := "FALSE",
                          O_Alarm => #AC_KeepPos5,
                          O_AlarmDisabled => "NotUsedBool",
                          O_AlarmABCondition => "NotUsedBool",
                          H_IAnim => #NotUsedH_HMI.H_IAnim);
   END_IF;
END_REGION

REGION Network 51: **** 2.2 - Alarms - Alarm Generation **** Reference Mode is active
   #AD_ReferencingActive := #ReferencingMode;
END_REGION

REGION Network 52: **** 2.2 - Alarms - Alarm Generation **** No bus control
   #AA_NoBusControl := #PODataNotEnabled AND #C_Config.EnableAlarmHW;
END_REGION

REGION Network 53: **** 2.2 - Alarms - Alarm Generation **** Flinta in Referencing Mode / **** 2.2 - Alarms - Alarm Generation **** Shuttle in Referencing Mode
   IF #IO_Modes.LMode.AlarmResetPB OR NOT #ReferencingMode THEN
       #AB_ReferencingMode := FALSE;   // RS flip-flop
   END_IF;
   IF #ReferencingMode THEN #AB_ReferencingMode := TRUE; END_IF;
END_REGION

REGION Network 54: **** 2.2 - Alarms - Alarm Generation **** The referencing of the Shuttle is not done
   #AB_NoReferencing := #H_ReferencingPos = 0;
END_REGION

REGION Network 55: **** 4.3 - Machine status - Operator Selection **** Manual request position 1
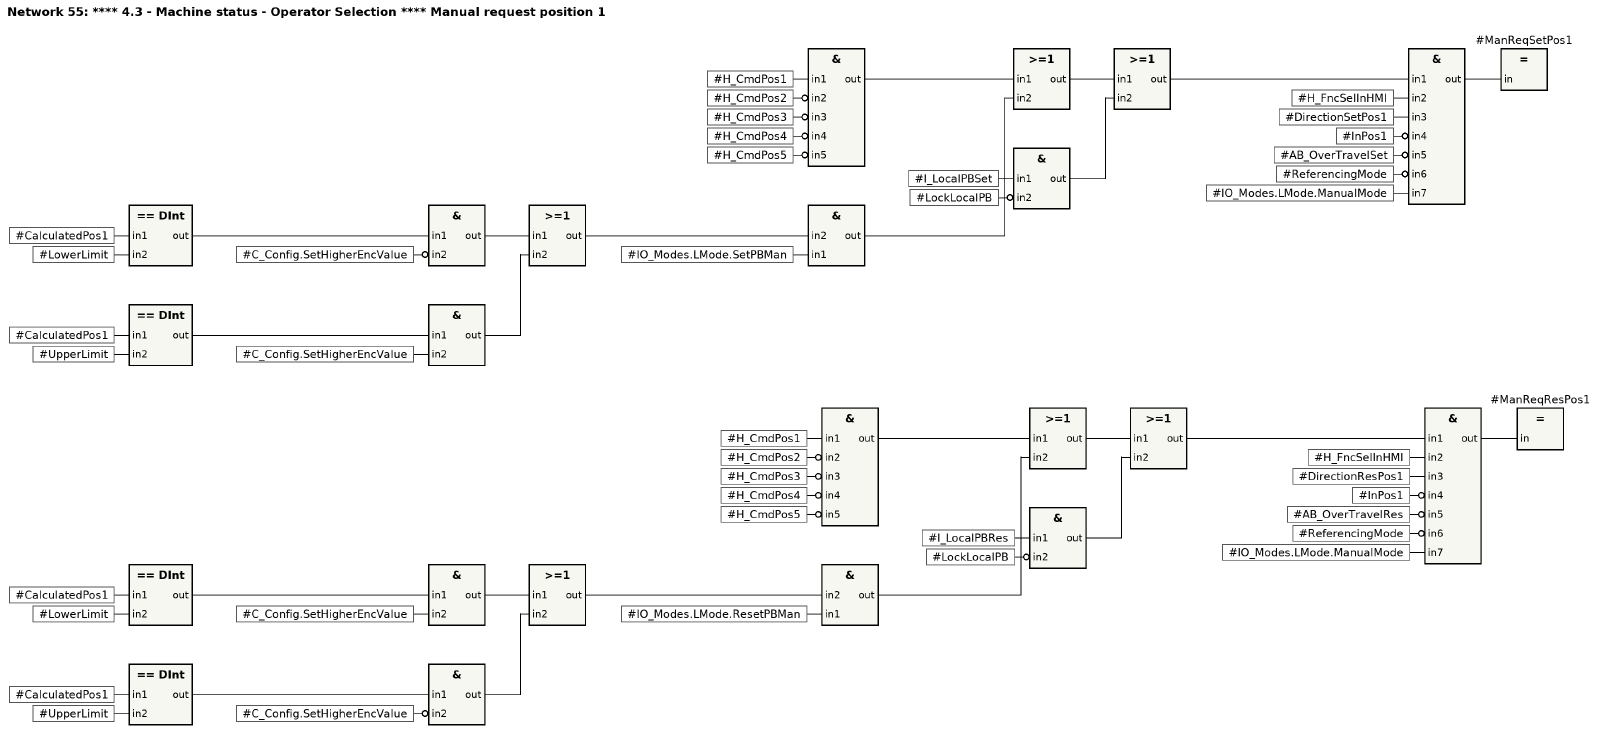
   #ManReqSetPos1 := ((#H_CmdPos1 AND NOT #H_CmdPos2 AND NOT #H_CmdPos3 AND NOT #H_CmdPos4 AND NOT #H_CmdPos5) OR ((((#CalculatedPos1 = #LowerLimit) AND NOT #C_Config.SetHigherEncValue) OR ((#CalculatedPos1 = #UpperLimit) AND #C_Config.SetHigherEncValue)) AND #IO_Modes.LMode.SetPBMan) OR (#I_LocalPBSet AND NOT #LockLocalPB)) AND #H_FncSelInHMI AND #DirectionSetPos1 AND NOT #InPos1 AND NOT #AB_OverTravelSet AND NOT #ReferencingMode AND #IO_Modes.LMode.ManualMode;
   #ManReqResPos1 := ((#H_CmdPos1 AND NOT #H_CmdPos2 AND NOT #H_CmdPos3 AND NOT #H_CmdPos4 AND NOT #H_CmdPos5) OR ((((#CalculatedPos1 = #LowerLimit) AND #C_Config.SetHigherEncValue) OR ((#CalculatedPos1 = #UpperLimit) AND NOT #C_Config.SetHigherEncValue)) AND #IO_Modes.LMode.ResetPBMan) OR (#I_LocalPBRes AND NOT #LockLocalPB)) AND #H_FncSelInHMI AND #DirectionResPos1 AND NOT #InPos1 AND NOT #AB_OverTravelRes AND NOT #ReferencingMode AND #IO_Modes.LMode.ManualMode;
END_REGION

REGION Network 56: **** 4.3 - Machine status - Operator Selection **** Manual request position 2
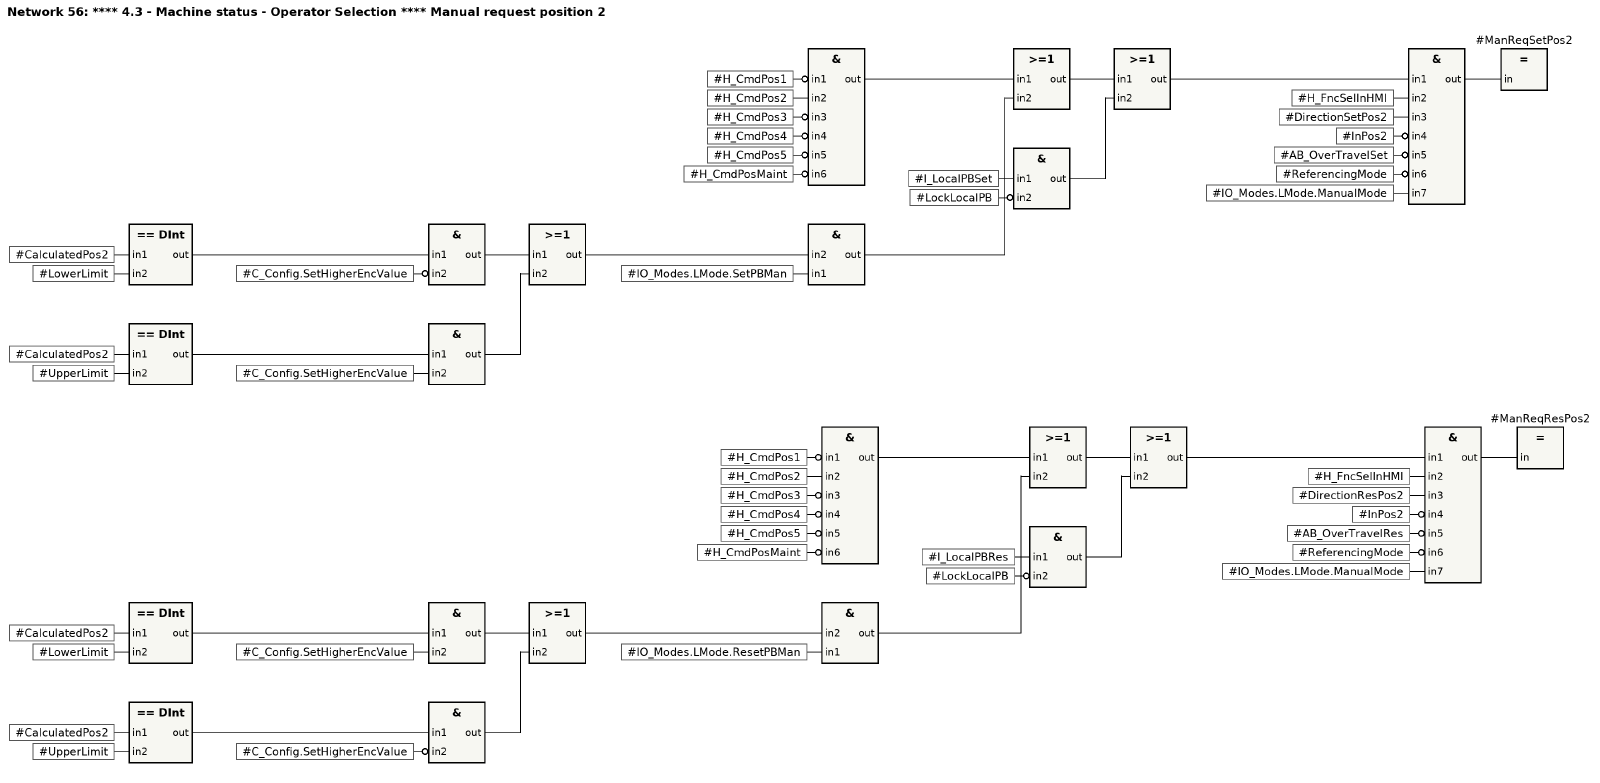
   #ManReqSetPos2 := ((NOT #H_CmdPos1 AND #H_CmdPos2 AND NOT #H_CmdPos3 AND NOT #H_CmdPos4 AND NOT #H_CmdPos5 AND NOT #H_CmdPosMaint) OR ((((#CalculatedPos2 = #LowerLimit) AND NOT #C_Config.SetHigherEncValue) OR ((#CalculatedPos2 = #UpperLimit) AND #C_Config.SetHigherEncValue)) AND #IO_Modes.LMode.SetPBMan) OR (#I_LocalPBSet AND NOT #LockLocalPB)) AND #H_FncSelInHMI AND #DirectionSetPos2 AND NOT #InPos2 AND NOT #AB_OverTravelSet AND NOT #ReferencingMode AND #IO_Modes.LMode.ManualMode;
   #ManReqResPos2 := ((NOT #H_CmdPos1 AND #H_CmdPos2 AND NOT #H_CmdPos3 AND NOT #H_CmdPos4 AND NOT #H_CmdPos5 AND NOT #H_CmdPosMaint) OR ((((#CalculatedPos2 = #LowerLimit) AND #C_Config.SetHigherEncValue) OR ((#CalculatedPos2 = #UpperLimit) AND NOT #C_Config.SetHigherEncValue)) AND #IO_Modes.LMode.ResetPBMan) OR (#I_LocalPBRes AND NOT #LockLocalPB)) AND #H_FncSelInHMI AND #DirectionResPos2 AND NOT #InPos2 AND NOT #AB_OverTravelRes AND NOT #ReferencingMode AND #IO_Modes.LMode.ManualMode;
END_REGION

REGION Network 57: **** 4.3 - Machine status - Operator Selection **** Manual request position 3
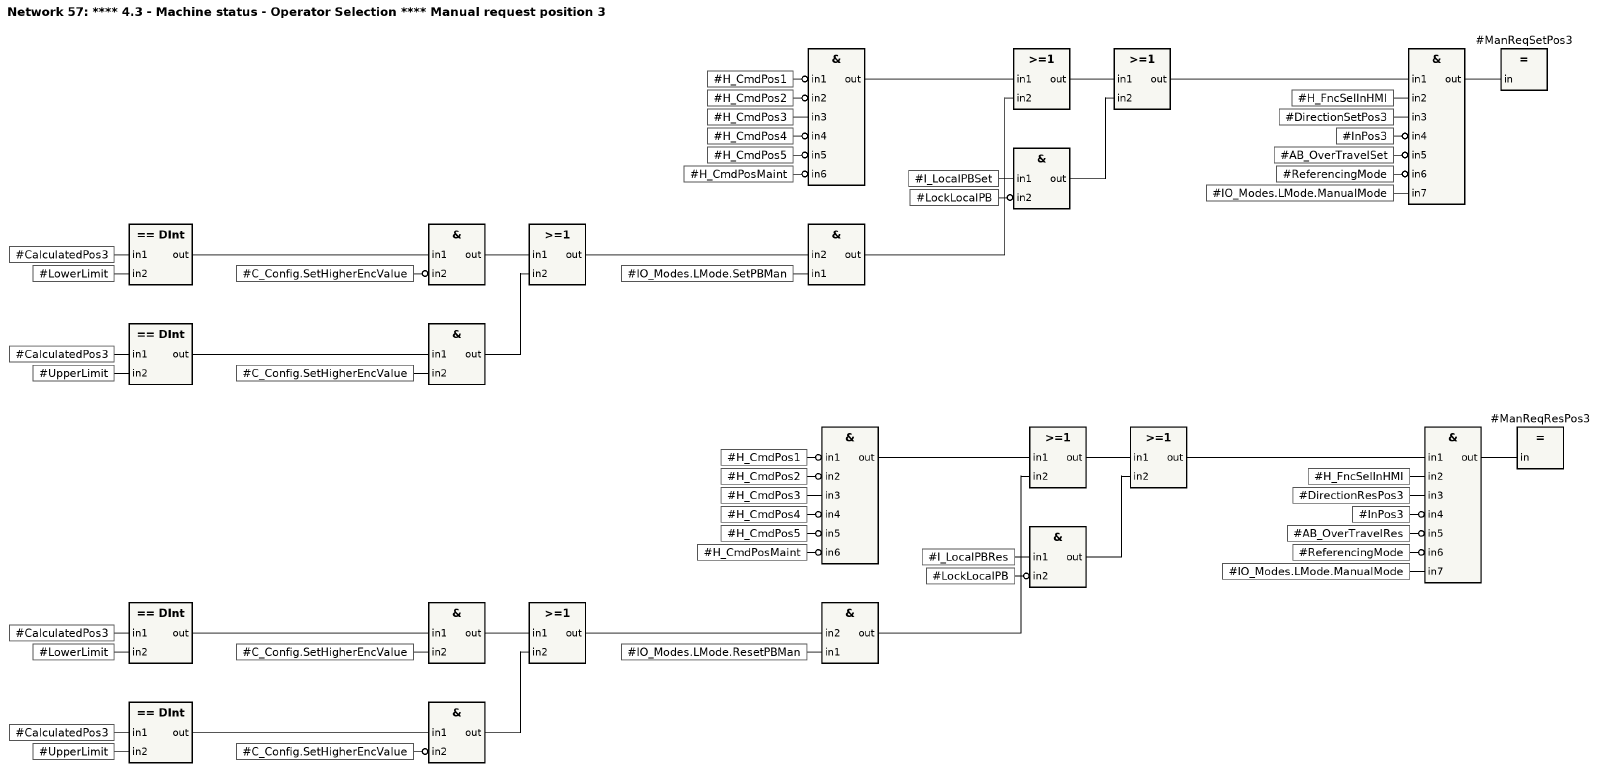
   #ManReqSetPos3 := ((NOT #H_CmdPos1 AND NOT #H_CmdPos2 AND #H_CmdPos3 AND NOT #H_CmdPos4 AND NOT #H_CmdPos5 AND NOT #H_CmdPosMaint) OR ((((#CalculatedPos3 = #LowerLimit) AND NOT #C_Config.SetHigherEncValue) OR ((#CalculatedPos3 = #UpperLimit) AND #C_Config.SetHigherEncValue)) AND #IO_Modes.LMode.SetPBMan) OR (#I_LocalPBSet AND NOT #LockLocalPB)) AND #H_FncSelInHMI AND #DirectionSetPos3 AND NOT #InPos3 AND NOT #AB_OverTravelSet AND NOT #ReferencingMode AND #IO_Modes.LMode.ManualMode;
   #ManReqResPos3 := ((NOT #H_CmdPos1 AND NOT #H_CmdPos2 AND #H_CmdPos3 AND NOT #H_CmdPos4 AND NOT #H_CmdPos5 AND NOT #H_CmdPosMaint) OR ((((#CalculatedPos3 = #LowerLimit) AND #C_Config.SetHigherEncValue) OR ((#CalculatedPos3 = #UpperLimit) AND NOT #C_Config.SetHigherEncValue)) AND #IO_Modes.LMode.ResetPBMan) OR (#I_LocalPBRes AND NOT #LockLocalPB)) AND #H_FncSelInHMI AND #DirectionResPos3 AND NOT #InPos3 AND NOT #AB_OverTravelRes AND NOT #ReferencingMode AND #IO_Modes.LMode.ManualMode;
END_REGION

REGION Network 58: **** 4.3 - Machine status - Operator Selection **** Manual request position 4
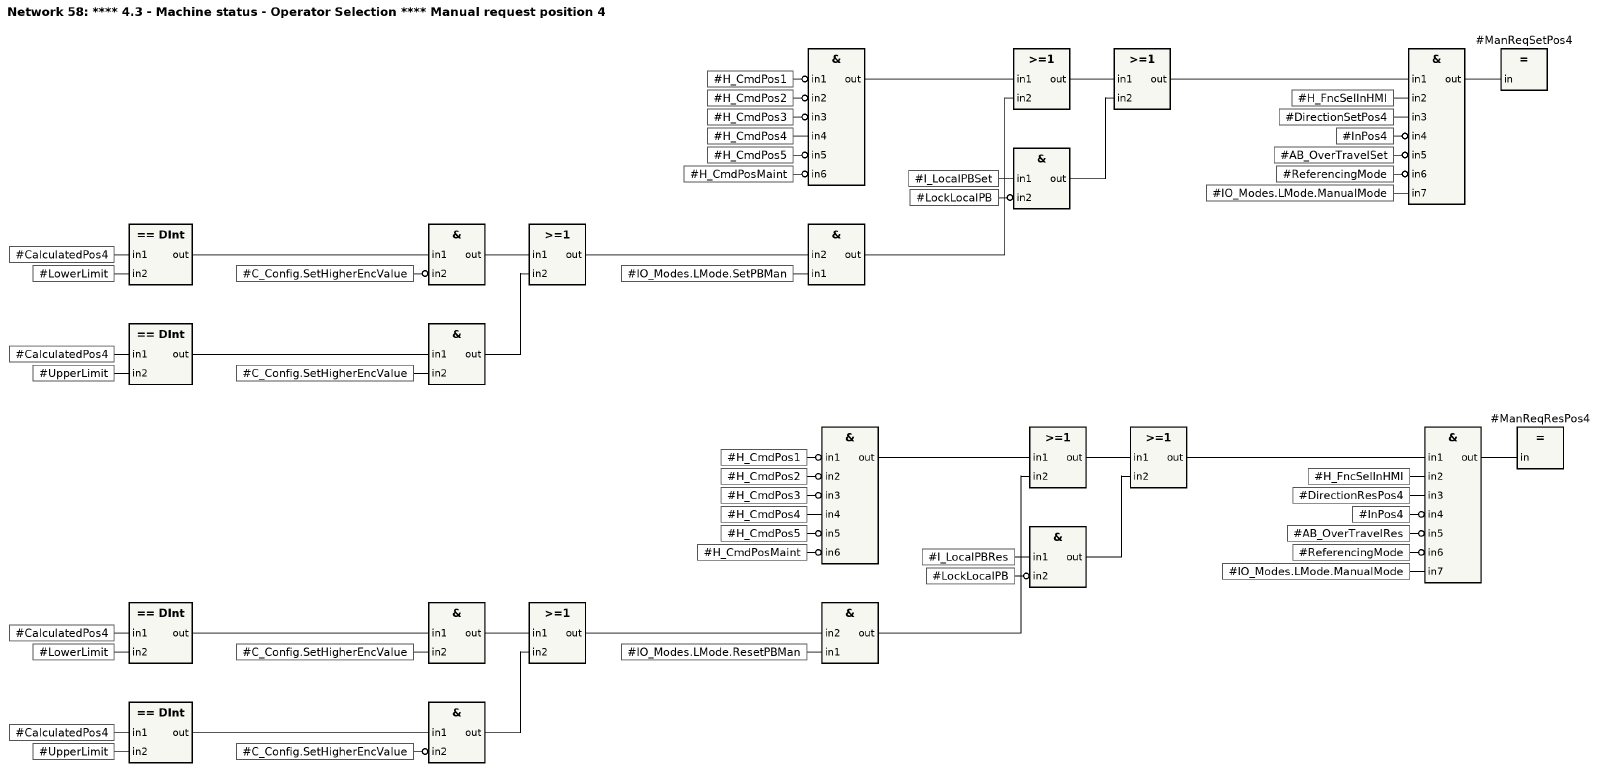
   #ManReqSetPos4 := ((NOT #H_CmdPos1 AND NOT #H_CmdPos2 AND NOT #H_CmdPos3 AND #H_CmdPos4 AND NOT #H_CmdPos5 AND NOT #H_CmdPosMaint) OR ((((#CalculatedPos4 = #LowerLimit) AND NOT #C_Config.SetHigherEncValue) OR ((#CalculatedPos4 = #UpperLimit) AND #C_Config.SetHigherEncValue)) AND #IO_Modes.LMode.SetPBMan) OR (#I_LocalPBSet AND NOT #LockLocalPB)) AND #H_FncSelInHMI AND #DirectionSetPos4 AND NOT #InPos4 AND NOT #AB_OverTravelSet AND NOT #ReferencingMode AND #IO_Modes.LMode.ManualMode;
   #ManReqResPos4 := ((NOT #H_CmdPos1 AND NOT #H_CmdPos2 AND NOT #H_CmdPos3 AND #H_CmdPos4 AND NOT #H_CmdPos5 AND NOT #H_CmdPosMaint) OR ((((#CalculatedPos4 = #LowerLimit) AND #C_Config.SetHigherEncValue) OR ((#CalculatedPos4 = #UpperLimit) AND NOT #C_Config.SetHigherEncValue)) AND #IO_Modes.LMode.ResetPBMan) OR (#I_LocalPBRes AND NOT #LockLocalPB)) AND #H_FncSelInHMI AND #DirectionResPos4 AND NOT #InPos4 AND NOT #AB_OverTravelRes AND NOT #ReferencingMode AND #IO_Modes.LMode.ManualMode;
END_REGION

REGION Network 59: **** 4.3 - Machine status - Operator Selection **** Manual request position 5
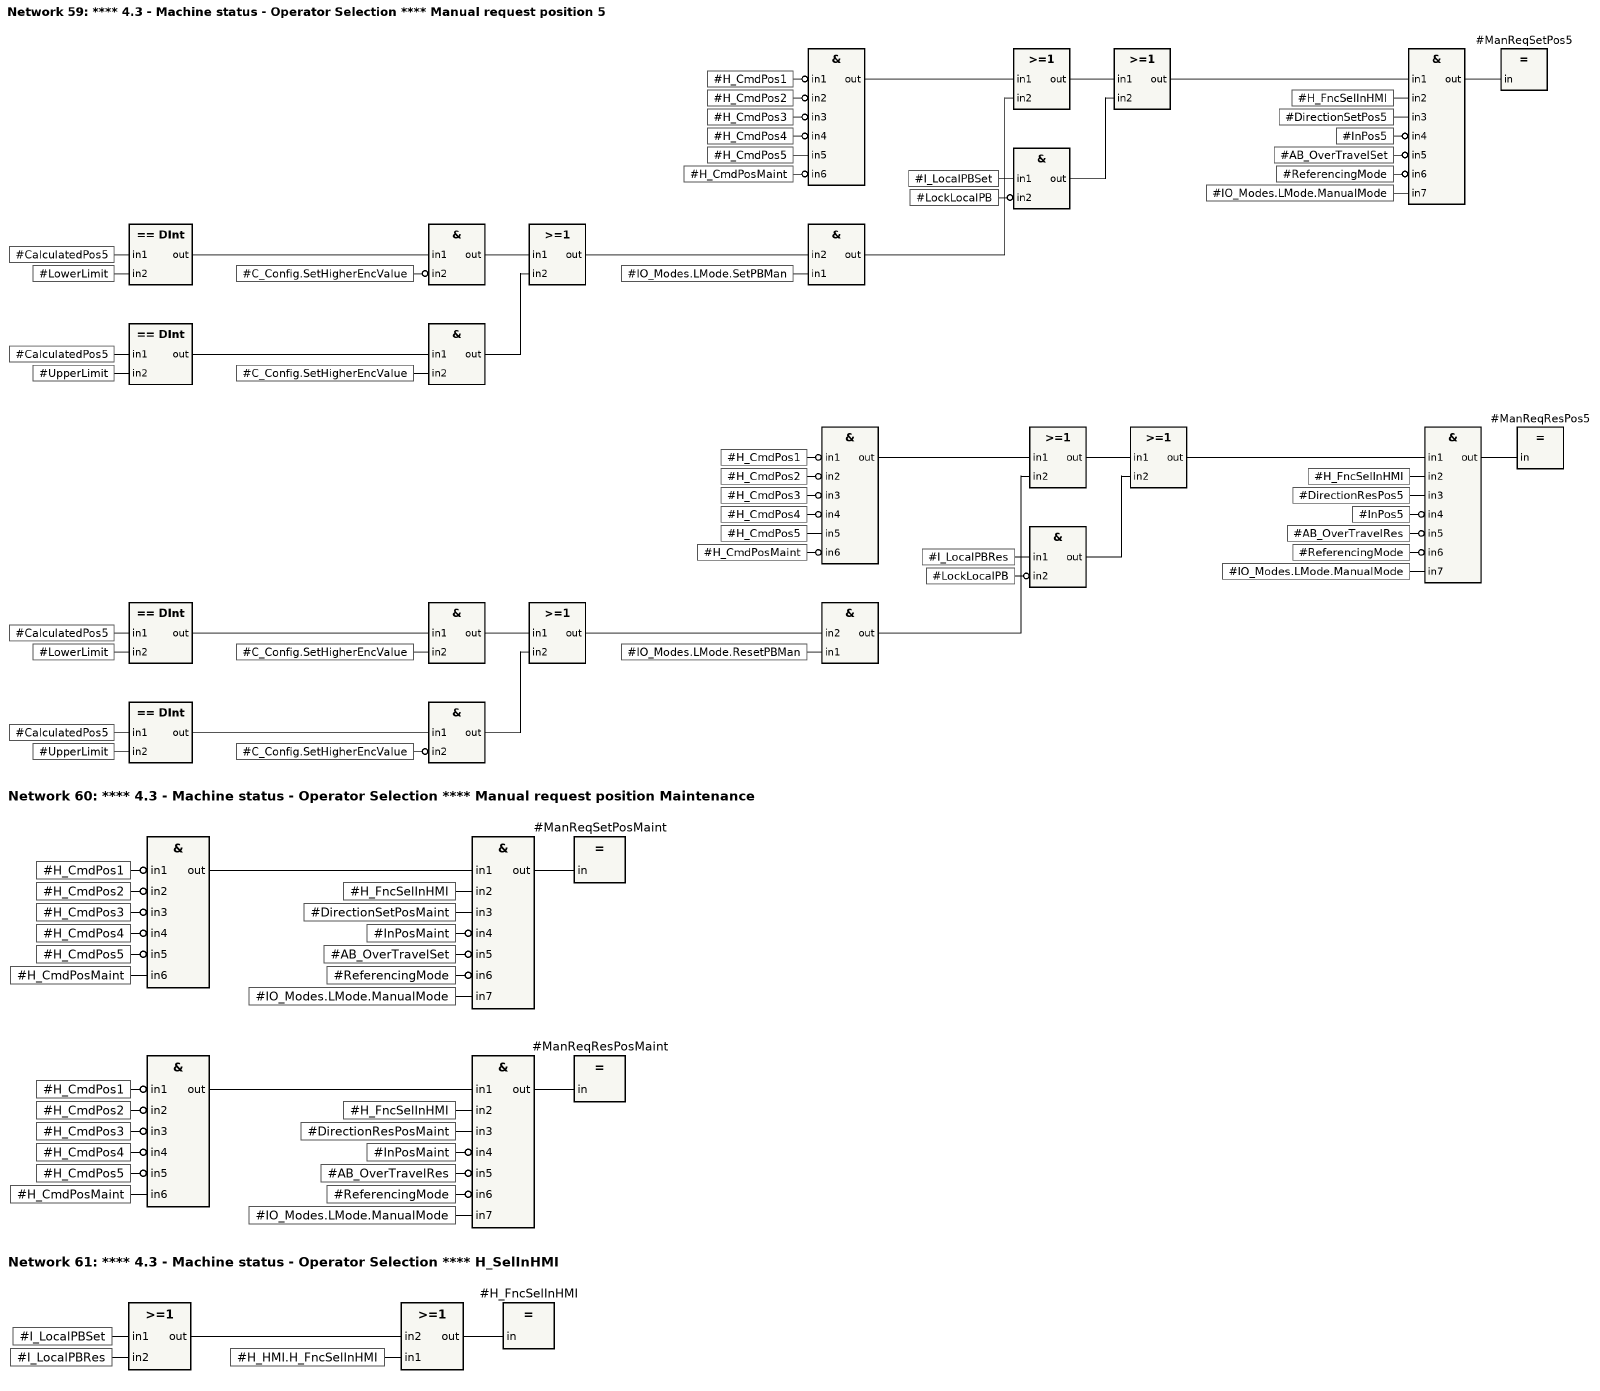
   #ManReqSetPos5 := ((NOT #H_CmdPos1 AND NOT #H_CmdPos2 AND NOT #H_CmdPos3 AND NOT #H_CmdPos4 AND #H_CmdPos5 AND NOT #H_CmdPosMaint) OR ((((#CalculatedPos5 = #LowerLimit) AND NOT #C_Config.SetHigherEncValue) OR ((#CalculatedPos5 = #UpperLimit) AND #C_Config.SetHigherEncValue)) AND #IO_Modes.LMode.SetPBMan) OR (#I_LocalPBSet AND NOT #LockLocalPB)) AND #H_FncSelInHMI AND #DirectionSetPos5 AND NOT #InPos5 AND NOT #AB_OverTravelSet AND NOT #ReferencingMode AND #IO_Modes.LMode.ManualMode;
   #ManReqResPos5 := ((NOT #H_CmdPos1 AND NOT #H_CmdPos2 AND NOT #H_CmdPos3 AND NOT #H_CmdPos4 AND #H_CmdPos5 AND NOT #H_CmdPosMaint) OR ((((#CalculatedPos5 = #LowerLimit) AND #C_Config.SetHigherEncValue) OR ((#CalculatedPos5 = #UpperLimit) AND NOT #C_Config.SetHigherEncValue)) AND #IO_Modes.LMode.ResetPBMan) OR (#I_LocalPBRes AND NOT #LockLocalPB)) AND #H_FncSelInHMI AND #DirectionResPos5 AND NOT #InPos5 AND NOT #AB_OverTravelRes AND NOT #ReferencingMode AND #IO_Modes.LMode.ManualMode;
END_REGION

REGION Network 60: **** 4.3 - Machine status - Operator Selection **** Manual request position Maintenance
   #ManReqSetPosMaint := NOT #H_CmdPos1 AND NOT #H_CmdPos2 AND NOT #H_CmdPos3 AND NOT #H_CmdPos4 AND NOT #H_CmdPos5 AND #H_CmdPosMaint AND #H_FncSelInHMI AND #DirectionSetPosMaint AND NOT #InPosMaint AND NOT #AB_OverTravelSet AND NOT #ReferencingMode AND #IO_Modes.LMode.ManualMode;
   #ManReqResPosMaint := NOT #H_CmdPos1 AND NOT #H_CmdPos2 AND NOT #H_CmdPos3 AND NOT #H_CmdPos4 AND NOT #H_CmdPos5 AND #H_CmdPosMaint AND #H_FncSelInHMI AND #DirectionResPosMaint AND NOT #InPosMaint AND NOT #AB_OverTravelRes AND NOT #ReferencingMode AND #IO_Modes.LMode.ManualMode;
END_REGION

REGION Network 61: **** 4.3 - Machine status - Operator Selection **** H_SelInHMI
   #H_FncSelInHMI := #I_LocalPBSet OR #I_LocalPBRes OR #H_HMI.H_FncSelInHMI;
END_REGION

REGION Network 62: **** 4.3 - Machine status - Operator Selection **** Reset H_SelInHMI
   // Reset H_SelInHMI
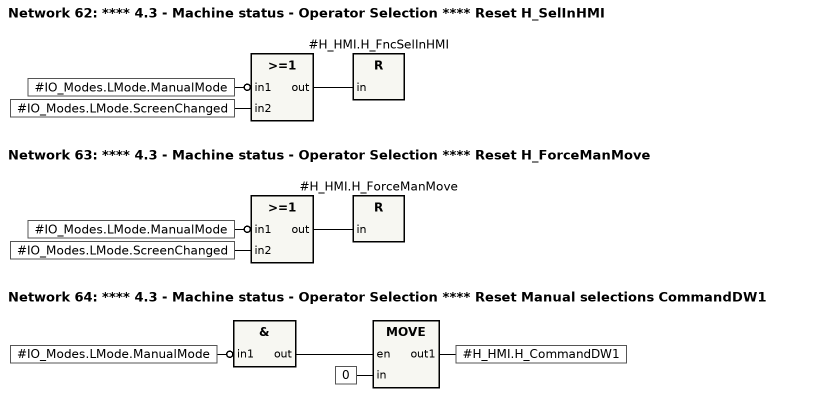
   IF NOT #IO_Modes.LMode.ManualMode OR #IO_Modes.LMode.ScreenChanged THEN
       #H_HMI.H_FncSelInHMI := FALSE;
   END_IF;
END_REGION

REGION Network 63: **** 4.3 - Machine status - Operator Selection **** Reset H_ForceManMove
   // Reset H_ForceManMove
   IF NOT #IO_Modes.LMode.ManualMode OR #IO_Modes.LMode.ScreenChanged THEN
       #H_HMI.H_ForceManMove := FALSE;
   END_IF;
END_REGION

REGION Network 64: **** 4.3 - Machine status - Operator Selection **** Reset Manual selections CommandDW1
   // Reset all selections in the HMI
   IF NOT #IO_Modes.LMode.ManualMode THEN #H_HMI.H_CommandDW1 := 0; END_IF;
END_REGION

REGION Network 65: **** 4.4 - Machine status - Calculation **** Lower limit position
   // Calculate minimum value of all positions
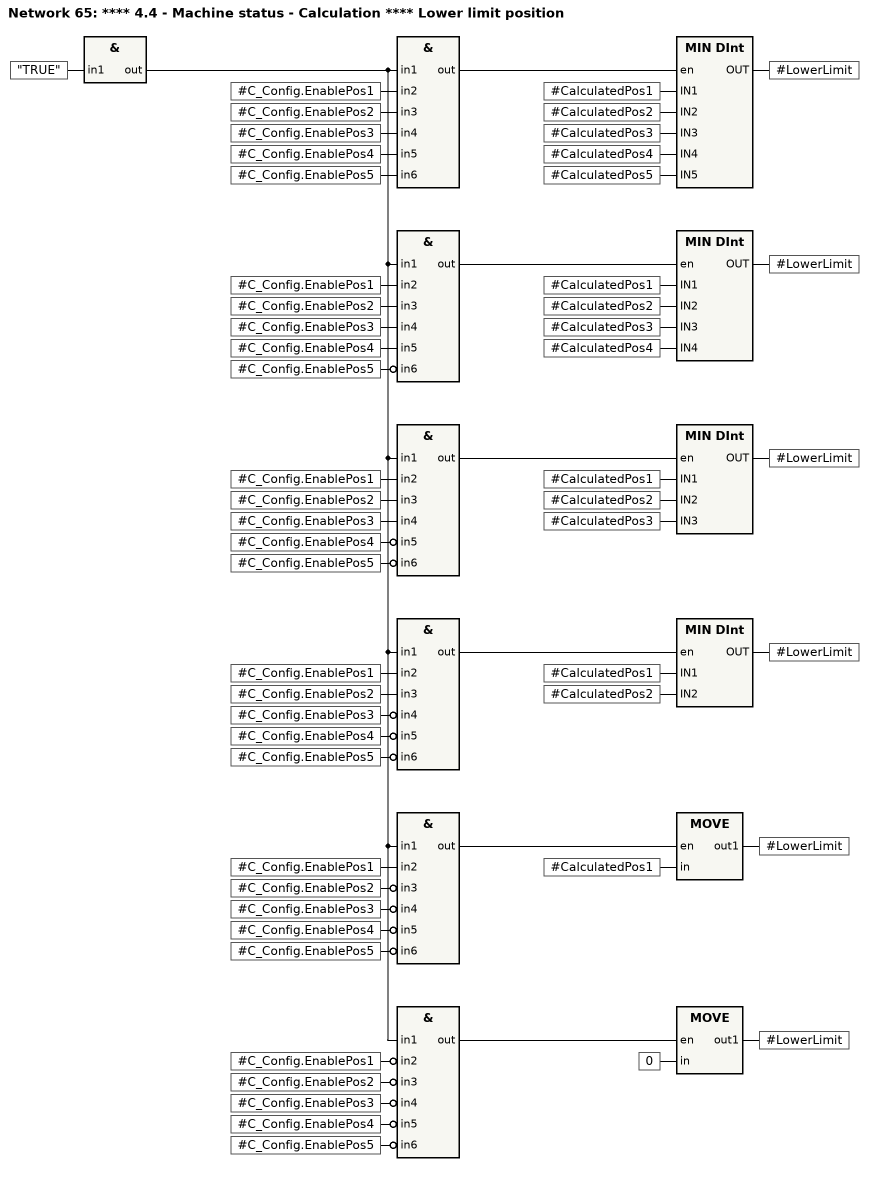
   IF "TRUE" AND #C_Config.EnablePos1 AND #C_Config.EnablePos2 AND #C_Config.EnablePos3 AND #C_Config.EnablePos4 AND #C_Config.EnablePos5 THEN
       #LowerLimit := MIN(IN1 := #CalculatedPos1, IN2 := #CalculatedPos2, IN3 := #CalculatedPos3, IN4 := #CalculatedPos4, IN5 := #CalculatedPos5);
   END_IF;
   IF "TRUE" AND #C_Config.EnablePos1 AND #C_Config.EnablePos2 AND #C_Config.EnablePos3 AND #C_Config.EnablePos4 AND NOT #C_Config.EnablePos5 THEN
       #LowerLimit := MIN(IN1 := #CalculatedPos1, IN2 := #CalculatedPos2, IN3 := #CalculatedPos3, IN4 := #CalculatedPos4);
   END_IF;
   IF "TRUE" AND #C_Config.EnablePos1 AND #C_Config.EnablePos2 AND #C_Config.EnablePos3 AND NOT #C_Config.EnablePos4 AND NOT #C_Config.EnablePos5 THEN
       #LowerLimit := MIN(IN1 := #CalculatedPos1, IN2 := #CalculatedPos2, IN3 := #CalculatedPos3);
   END_IF;
   IF "TRUE" AND #C_Config.EnablePos1 AND #C_Config.EnablePos2 AND NOT #C_Config.EnablePos3 AND NOT #C_Config.EnablePos4 AND NOT #C_Config.EnablePos5 THEN
       #LowerLimit := MIN(IN1 := #CalculatedPos1, IN2 := #CalculatedPos2);
   END_IF;
   IF "TRUE" AND #C_Config.EnablePos1 AND NOT #C_Config.EnablePos2 AND NOT #C_Config.EnablePos3 AND NOT #C_Config.EnablePos4 AND NOT #C_Config.EnablePos5 THEN
       #LowerLimit := #CalculatedPos1;
   END_IF;
   IF "TRUE" AND NOT #C_Config.EnablePos1 AND NOT #C_Config.EnablePos2 AND NOT #C_Config.EnablePos3 AND NOT #C_Config.EnablePos4 AND NOT #C_Config.EnablePos5 THEN
       #LowerLimit := 0;
   END_IF;
END_REGION

REGION Network 66: **** 4.4 - Machine status - Calculation **** Upper limit position
   // Calculate maximum value of all positions
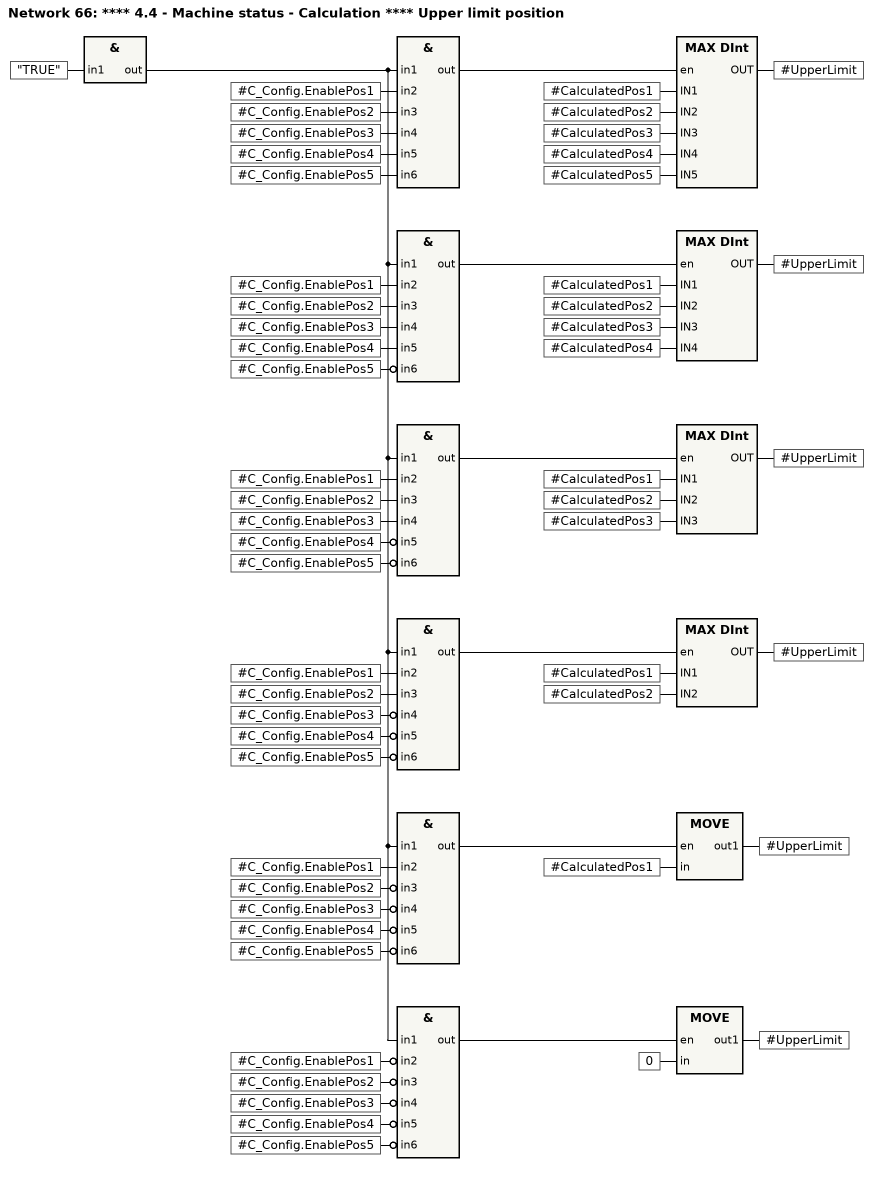
   IF "TRUE" AND #C_Config.EnablePos1 AND #C_Config.EnablePos2 AND #C_Config.EnablePos3 AND #C_Config.EnablePos4 AND #C_Config.EnablePos5 THEN
       #UpperLimit := MAX(IN1 := #CalculatedPos1, IN2 := #CalculatedPos2, IN3 := #CalculatedPos3, IN4 := #CalculatedPos4, IN5 := #CalculatedPos5);
   END_IF;
   IF "TRUE" AND #C_Config.EnablePos1 AND #C_Config.EnablePos2 AND #C_Config.EnablePos3 AND #C_Config.EnablePos4 AND NOT #C_Config.EnablePos5 THEN
       #UpperLimit := MAX(IN1 := #CalculatedPos1, IN2 := #CalculatedPos2, IN3 := #CalculatedPos3, IN4 := #CalculatedPos4);
   END_IF;
   IF "TRUE" AND #C_Config.EnablePos1 AND #C_Config.EnablePos2 AND #C_Config.EnablePos3 AND NOT #C_Config.EnablePos4 AND NOT #C_Config.EnablePos5 THEN
       #UpperLimit := MAX(IN1 := #CalculatedPos1, IN2 := #CalculatedPos2, IN3 := #CalculatedPos3);
   END_IF;
   IF "TRUE" AND #C_Config.EnablePos1 AND #C_Config.EnablePos2 AND NOT #C_Config.EnablePos3 AND NOT #C_Config.EnablePos4 AND NOT #C_Config.EnablePos5 THEN
       #UpperLimit := MAX(IN1 := #CalculatedPos1, IN2 := #CalculatedPos2);
   END_IF;
   IF "TRUE" AND #C_Config.EnablePos1 AND NOT #C_Config.EnablePos2 AND NOT #C_Config.EnablePos3 AND NOT #C_Config.EnablePos4 AND NOT #C_Config.EnablePos5 THEN
       #UpperLimit := #CalculatedPos1;
   END_IF;
   IF "TRUE" AND NOT #C_Config.EnablePos1 AND NOT #C_Config.EnablePos2 AND NOT #C_Config.EnablePos3 AND NOT #C_Config.EnablePos4 AND NOT #C_Config.EnablePos5 THEN
       #UpperLimit := 0;
   END_IF;
END_REGION

REGION Network 67: **** 4.6 - Machine Status - Indication **** Stop Detection set / **** 4.6 - Machine Status - Indication **** Reference Detection
   // Stop Detection set
